(* CODESYS project LuPumping_v3_42.project

Project tree, tasks and I/O mapping:
  LocalDevice : CODESYS Control for Raspberry Pi SL, 3S - Smart Software Solutions GmbH, version 3.5.16.0
    application Application
      libraries: Standard, * (System); VisuDialogs, * (System); SysMem, * (System); SysTimeRtc, * (System); SysRtc23, 3.5.13.0 (System); BASIC, * (OSCAT); CmpBitmapPool, * (System); Util, * (System)
      task VISU_TASK (cyclic, interval 4 ms, priority 31) calls VisuElems.Visu_Prg
      task EtherCAT_Task (cyclic, interval t#4ms, priority 1) calls EtherCAT_Master.EtherCAT_Task
      task MAIN (cyclic, interval t#20ms, priority 1) calls PLC_PRG
      global variables GVL
      Symbols
      Visu_Pages/
        visualisation Visualization_10
        visualisation Visualization_30
        visualisation Visualization_20
        visualisation Visualization_11
        image pool ImagePool
        visualisation Visualization_40
        image pool ImagePool_Presets
        visualisation Visualization_31
      Struct/
        data type ST_ControllerData
        data type ST_ModbusRegister
        data type ST_EtherCATData
        data type ST_PumpingData
        data type ST_PumpingData_HMI
        data type ST_PresetLU
        data type ST_OutBuffer
      program PLC_PRG [ST]
      program _00_Initialization [ST]
      program _01_Comms [ST]
      program _02_Ctrl [ST]
      program _03_daq_setup [ST]
      program _04_daq_input [ST]
      program _05_daq_output [ST]
      program _06_hmi [ST]
    I²C
    GPIOs_A_B : GPIOs A/B, 3S - Smart Software Solutions GmbH, version 3.5.11.0 (disabled)
        unmapped channels: digital inputs (GPIO0..GPIO31), digital outputs (GPIO0..GPIO31)
    SPI
    EtherCAT_Master : EtherCAT Master, 3S - Smart Software Solutions GmbH, version 3.5.16.0
        settings: NetworkName = 'eth0'; NetworkName = "eth0"; SelectNetworkByName = True; SrcAddress1 = 47143; SrcAddress2 = 3947725782
      EK1101 : EK1101 EtherCAT Coupler (2A E-Bus, ID switch), Beckhoff Automation GmbH & Co. KG, order no. EK1101, version Revision=16#00120000
          settings: StationAlias = 0
          unmapped channels: ID
        EL2502_3 : EL2502 2Ch. PWM output, 24V, Beckhoff Automation GmbH & Co. KG, order no. EL2502, version Revision=16#001A0000
            settings: StationAlias = 0
            output Application.GVL.EthCAT.PumpPWM_INT16[5] : UINT  // PWM output
            output Application.GVL.EthCAT.PumpPWM_INT16[6] : UINT  // PWM output
        EL2502_1 : EL2502 2Ch. PWM output, 24V, Beckhoff Automation GmbH & Co. KG, order no. EL2502, version Revision=16#001A0000
            settings: StationAlias = 0; RxTxPdo.NumberofExcludes = 2; RxTxPdo.NumberofEntries = 1; RxTxPdo.Index = 16#1600; RxTxPdo.Fixed = True; RxTxPdo.Mandatory = False; RxTxPdo.Virtual = False; RxTxPdo.Sm = 2; RxTxPdo.Su = 2; RxTxPdo.Name = 'PWM Outputs Channel 1'; RxTxPdo.DependOnSlot = False; RxTxPdo.DependOnSlotGroup = False; RxTxPdo.OverwrittenByModule = False; Exclude = [16#1602,16#1604]; PWM output.Index = 16#7000; PWM output.SubIndex = 17; PWM output.Size = 16; PWM output.Offset = 0; PWM output.DependOnSlot = False; PWM output.DependOnSlotGroup = False; RxTxPdo.NumberofExcludes = 2; RxTxPdo.NumberofEntries = 1; RxTxPdo.Index = 16#1601; RxTxPdo.Fixed = True; RxTxPdo.Mandatory = False; RxTxPdo.Virtual = False; RxTxPdo.Sm = 2; RxTxPdo.Su = 2; RxTxPdo.Name = 'PWM Outputs Channel 2'; RxTxPdo.DependOnSlot = False; RxTxPdo.DependOnSlotGroup = False; RxTxPdo.OverwrittenByModule = False; Exclude = [16#1603,16#1605]; PWM output.Index = 16#7010; PWM output.SubIndex = 17; PWM output.Size = 16; PWM output.Offset = 0; PWM output.DependOnSlot = False; PWM output.DependOnSlotGroup = False; RxTxPdo.NumberofExcludes = 2;
              RxTxPdo.NumberofEntries = 2; RxTxPdo.Index = 16#1602; RxTxPdo.Fixed = True; RxTxPdo.Mandatory = False; RxTxPdo.Virtual = False; RxTxPdo.Sm = -1; RxTxPdo.Su = -1; RxTxPdo.Name = 'PWM Outputs Channel 1'; RxTxPdo.DependOnSlot = False; RxTxPdo.DependOnSlotGroup = False; RxTxPdo.OverwrittenByModule = False; Exclude = [16#1600,16#1604]; PWM output.Index = 16#7000; PWM output.SubIndex = 17; PWM output.Size = 16; PWM output.Offset = 0; PWM output.DependOnSlot = False; PWM output.DependOnSlotGroup = False; PWM period.Index = 16#7000; PWM period.SubIndex = 18; PWM period.Size = 16; PWM period.Offset = 0; PWM period.DependOnSlot = False; PWM period.DependOnSlotGroup = False; RxTxPdo.NumberofExcludes = 2; RxTxPdo.NumberofEntries = 2; RxTxPdo.Index = 16#1603; RxTxPdo.Fixed = True; RxTxPdo.Mandatory = False; RxTxPdo.Virtual = False; RxTxPdo.Sm = -1; RxTxPdo.Su = -1; RxTxPdo.Name = 'PWM Outputs Channel 2'; RxTxPdo.DependOnSlot = False; RxTxPdo.DependOnSlotGroup = False; RxTxPdo.OverwrittenByModule = False; Exclude = [16#1601,16#1605]; PWM output.Index = 16#7010; PWM output.SubIndex = 17; PWM output.Size = 16;
              PWM output.Offset = 0; PWM output.DependOnSlot = False; PWM output.DependOnSlotGroup = False; PWM period.Index = 16#7010; PWM period.SubIndex = 18; PWM period.Size = 16; PWM period.Offset = 0; PWM period.DependOnSlot = False; PWM period.DependOnSlotGroup = False; RxTxPdo.NumberofExcludes = 2; RxTxPdo.NumberofEntries = 2; RxTxPdo.Index = 16#1604; RxTxPdo.Fixed = True; RxTxPdo.Mandatory = False; RxTxPdo.Virtual = False; RxTxPdo.Sm = -1; RxTxPdo.Su = -1; RxTxPdo.Name = 'PWM Outputs Channel 1'; RxTxPdo.DependOnSlot = False; RxTxPdo.DependOnSlotGroup = False; RxTxPdo.OverwrittenByModule = False; Exclude = [16#1600,16#1602]; PWM output.Index = 16#7000; PWM output.SubIndex = 17; PWM output.Size = 16; PWM output.Offset = 0; PWM output.DependOnSlot = False; PWM output.DependOnSlotGroup = False; PWM period 1Hz.Index = 16#7000; PWM period 1Hz.SubIndex = 19; PWM period 1Hz.Size = 32; PWM period 1Hz.Offset = 0; PWM period 1Hz.DependOnSlot = False; PWM period 1Hz.DependOnSlotGroup = False; RxTxPdo.NumberofExcludes = 2; RxTxPdo.NumberofEntries = 2; RxTxPdo.Index = 16#1605; RxTxPdo.Fixed = True; RxTxPdo.Mandatory = False; RxTxPdo.Virtual = False;
              RxTxPdo.Sm = -1; RxTxPdo.Su = -1; RxTxPdo.Name = 'PWM Outputs Channel 2'; RxTxPdo.DependOnSlot = False; RxTxPdo.DependOnSlotGroup = False; RxTxPdo.OverwrittenByModule = False; Exclude = [16#1601,16#1603]; PWM output.Index = 16#7010; PWM output.SubIndex = 17; PWM output.Size = 16; PWM output.Offset = 0; PWM output.DependOnSlot = False; PWM output.DependOnSlotGroup = False; PWM period 1Hz.Index = 16#7010; PWM period 1Hz.SubIndex = 19; PWM period 1Hz.Size = 32; PWM period 1Hz.Offset = 0; PWM period 1Hz.DependOnSlot = False; PWM period 1Hz.DependOnSlotGroup = False; PWM output.Name = 'PWM output'; PWM output.DataType = 'UINT'; PWM output.Default = ''; PWM output.Comment = ''; PWM output.Name = 'PWM output'; PWM output.DataType = 'UINT'; PWM output.Default = ''; PWM output.Comment = ''; PWM output.Name = 'PWM output'; PWM output.DataType = 'UINT'; PWM output.Default = ''; PWM output.Comment = ''; PWM period.Name = 'PWM period'; PWM period.DataType = 'UINT'; PWM period.Default = ''; PWM period.Comment = ''; PWM output.Name = 'PWM output'; PWM output.DataType = 'UINT'; PWM output.Default = ''; PWM output.Comment = ''; PWM period.Name = 'PWM period';
              PWM period.DataType = 'UINT'; PWM period.Default = ''; PWM period.Comment = ''; PWM output.Name = 'PWM output'; PWM output.DataType = 'UINT'; PWM output.Default = ''; PWM output.Comment = ''; PWM period 1Hz.Name = 'PWM period 1Hz'; PWM period 1Hz.DataType = 'UDINT'; PWM period 1Hz.Default = ''; PWM period 1Hz.Comment = ''; PWM output.Name = 'PWM output'; PWM output.DataType = 'UINT'; PWM output.Default = ''; PWM output.Comment = ''; PWM period 1Hz.Name = 'PWM period 1Hz'; PWM period 1Hz.DataType = 'UDINT'; PWM period 1Hz.Default = ''; PWM period 1Hz.Comment = ''
            output Application.GVL.EthCAT.PumpPWM_INT16[1] : UINT  // PWM output
            output Application.GVL.EthCAT.PumpPWM_INT16[2] : UINT  // PWM output
        EL2502_2 : EL2502 2Ch. PWM output, 24V, Beckhoff Automation GmbH & Co. KG, order no. EL2502, version Revision=16#001A0000
            settings: StationAlias = 0
            output Application.GVL.EthCAT.PumpPWM_INT16[3] : UINT  // PWM output
            output Application.GVL.EthCAT.PumpPWM_INT16[4] : UINT  // PWM output
        EL3048 : EL3048 8Ch. Ana. Input 0-20mA, Beckhoff Automation GmbH & Co. KG, order no. EL3048, version Revision=16#00140000
            settings: StationAlias = 0
            input  Application.GVL.EthCAT.Flow2_INT16[1] : INT  // Value
            input  Application.GVL.EthCAT.Flow2_INT16[2] : INT  // Value
            input  Application.GVL.EthCAT.Flow2_INT16[3] : INT  // Value
            input  Application.GVL.EthCAT.Conductivity_INT16 : INT  // Value
            input  Application.GVL.EthCAT.DeltaP2_INT16[1] : INT  // Value
            input  Application.GVL.EthCAT.DeltaP2_INT16[2] : INT  // Value
            unmapped channels: Status__Underrange, Status__Overrange, Status__Limit 1, Status__Limit 1, Status__Limit 2, Status__Limit 2, Status__Error, ---, ---, ---, ---, ---, ---, ---, Status__TxPDO State, Status__TxPDO Toggle, Status__Underrange, Status__Overrange, Status__Limit 1, Status__Limit 1, Status__Limit 2, Status__Limit 2, Status__Error, ---, ---, ---, ---, ---, ---, ---, Status__TxPDO State, Status__TxPDO Toggle, Status__Underrange, Status__Overrange, Status__Limit 1, Status__Limit 1, Status__Limit 2, Status__Limit 2, Status__Error, ---,
              ---, ---, ---, ---, ---, ---, Status__TxPDO State, Status__TxPDO Toggle, Status__Underrange, Status__Overrange, Status__Limit 1, Status__Limit 1, Status__Limit 2, Status__Limit 2, Status__Error, ---, ---, ---, ---, ---, ---, ---, Status__TxPDO State, Status__TxPDO Toggle, Status__Underrange, Status__Overrange, Status__Limit 1, Status__Limit 1, Status__Limit 2, Status__Limit 2, Status__Error, ---, ---, ---, ---, ---, ---, ---, Status__TxPDO State, Status__TxPDO Toggle,
              Status__Underrange, Status__Overrange, Status__Limit 1, Status__Limit 1, Status__Limit 2, Status__Limit 2, Status__Error, ---, ---, ---, ---, ---, ---, ---, Status__TxPDO State, Status__TxPDO Toggle, Status__Underrange, Status__Overrange, Status__Limit 1, Status__Limit 1, Status__Limit 2, Status__Limit 2, Status__Error, ---, ---, ---, ---, ---, ---, ---, Status__TxPDO State, Status__TxPDO Toggle, Value, Status__Underrange, Status__Overrange, Status__Limit 1, Status__Limit 1, Status__Limit 2, Status__Limit 2, Status__Error,
              ---, ---, ---, ---, ---, ---, ---, Status__TxPDO State, Status__TxPDO Toggle, Value
        EL4008 : EL4008 8Ch. Ana. Output 0-10V, 12bit, Beckhoff Automation GmbH & Co. KG, order no. EL4008, version Revision=16#00140000
            settings: StationAlias = 0
            output Application.GVL.EthCAT.ValveOD_INT16[1] : INT  // Analog output
            output Application.GVL.EthCAT.ValveOD_INT16[2] : INT  // Analog output
            output Application.GVL.EthCAT.VPPE_INT16 : INT  // Analog output
            output Application.GVL.EthCAT.ValveOD_INT16[3] : INT  // Analog output
            output Application.GVL.EthCAT.ValveOD_INT16[4] : INT  // Analog output
            unmapped channels: Analog output, Analog output, Analog output
        EL2008 : EL2008 8Ch. Dig. Output 24V, 0.5A, Beckhoff Automation GmbH & Co. KG, order no. EL2008, version Revision=16#00120000
            settings: StationAlias = 0
            output Application.GVL.EthCAT.Valve3_ON[1] : BIT  // Output
            output Application.GVL.EthCAT.Valve3_ON[2] : BIT  // Output
            output Application.GVL.EthCAT.Valve3_ON[3] : BIT  // Output
            output Application.GVL.EthCAT.Valve3_ON[4] : BIT  // Output
            output Application.GVL.EthCAT.Valve3_ON[5] : BIT  // Output
            output Application.GVL.EthCAT.Valve3_ON[6] : BIT  // Output
            output Application.GVL.EthCAT.Valve3_ON[7] : BIT  // Output
            output Application.GVL.EthCAT.Valve3_ON[8] : BIT  // Output
        EL2008_1 : EL2008 8Ch. Dig. Output 24V, 0.5A, Beckhoff Automation GmbH & Co. KG, order no. EL2008, version Revision=16#00120000
            settings: StationAlias = 0
            output Application.GVL.EthCAT.Valve3_ON[9] : BIT  // Output
            output Application.GVL.EthCAT.Valve3_ON[10] : BIT  // Output
            unmapped channels: Output, Output, Output, Output, Output, Output
        EL3068_1 : EL3068 8Ch. Ana. Input 0-10V, Beckhoff Automation GmbH & Co. KG, order no. EL3068, version Revision=16#00140000
            settings: StationAlias = 0
            input  Application.GVL.EthCAT.Temperature1_INT16[1] : INT  // Value
            input  Application.GVL.EthCAT.Pressure1_INT16[1] : INT  // Value
            input  Application.GVL.EthCAT.Temperature1_INT16[2] : INT  // Value
            input  Application.GVL.EthCAT.Pressure1_INT16[2] : INT  // Value
            input  Application.GVL.EthCAT.Temperature1_INT16[3] : INT  // Value
            input  Application.GVL.EthCAT.Pressure1_INT16[3] : INT  // Value
            input  Application.GVL.EthCAT.Temperature1_INT16[4] : INT  // Value
            input  Application.GVL.EthCAT.Pressure1_INT16[4] : INT  // Value
            unmapped channels: Status__Underrange, Status__Overrange, Status__Limit 1, Status__Limit 1, Status__Limit 2, Status__Limit 2, Status__Error, ---, ---, ---, ---, ---, ---, ---, Status__TxPDO State, Status__TxPDO Toggle, Status__Underrange, Status__Overrange, Status__Limit 1, Status__Limit 1, Status__Limit 2, Status__Limit 2, Status__Error, ---, ---, ---, ---, ---, ---, ---, Status__TxPDO State, Status__TxPDO Toggle, Status__Underrange, Status__Overrange, Status__Limit 1, Status__Limit 1, Status__Limit 2, Status__Limit 2, Status__Error, ---,
              ---, ---, ---, ---, ---, ---, Status__TxPDO State, Status__TxPDO Toggle, Status__Underrange, Status__Overrange, Status__Limit 1, Status__Limit 1, Status__Limit 2, Status__Limit 2, Status__Error, ---, ---, ---, ---, ---, ---, ---, Status__TxPDO State, Status__TxPDO Toggle, Status__Underrange, Status__Overrange, Status__Limit 1, Status__Limit 1, Status__Limit 2, Status__Limit 2, Status__Error, ---, ---, ---, ---, ---, ---, ---, Status__TxPDO State, Status__TxPDO Toggle,
              Status__Underrange, Status__Overrange, Status__Limit 1, Status__Limit 1, Status__Limit 2, Status__Limit 2, Status__Error, ---, ---, ---, ---, ---, ---, ---, Status__TxPDO State, Status__TxPDO Toggle, Status__Underrange, Status__Overrange, Status__Limit 1, Status__Limit 1, Status__Limit 2, Status__Limit 2, Status__Error, ---, ---, ---, ---, ---, ---, ---, Status__TxPDO State, Status__TxPDO Toggle, Status__Underrange, Status__Overrange, Status__Limit 1, Status__Limit 1, Status__Limit 2, Status__Limit 2, Status__Error, ---,
              ---, ---, ---, ---, ---, ---, Status__TxPDO State, Status__TxPDO Toggle
        EL3068 : EL3068 8Ch. Ana. Input 0-10V, Beckhoff Automation GmbH & Co. KG, order no. EL3068, version Revision=16#00140000
            settings: StationAlias = 0
            input  Application.GVL.EthCAT.Level_INT16[1] : INT  // Value
            input  Application.GVL.EthCAT.Level_INT16[2] : INT  // Value
            input  Application.GVL.EthCAT.Level_INT16[3] : INT  // Value
            input  Application.GVL.EthCAT.Level_INT16[4] : INT  // Value
            unmapped channels: Status__Underrange, Status__Overrange, Status__Limit 1, Status__Limit 1, Status__Limit 2, Status__Limit 2, Status__Error, ---, ---, ---, ---, ---, ---, ---, Status__TxPDO State, Status__TxPDO Toggle, Status__Underrange, Status__Overrange, Status__Limit 1, Status__Limit 1, Status__Limit 2, Status__Limit 2, Status__Error, ---, ---, ---, ---, ---, ---, ---, Status__TxPDO State, Status__TxPDO Toggle, Status__Underrange, Status__Overrange, Status__Limit 1, Status__Limit 1, Status__Limit 2, Status__Limit 2, Status__Error, ---,
              ---, ---, ---, ---, ---, ---, Status__TxPDO State, Status__TxPDO Toggle, Status__Underrange, Status__Overrange, Status__Limit 1, Status__Limit 1, Status__Limit 2, Status__Limit 2, Status__Error, ---, ---, ---, ---, ---, ---, ---, Status__TxPDO State, Status__TxPDO Toggle, Status__Underrange, Status__Overrange, Status__Limit 1, Status__Limit 1, Status__Limit 2, Status__Limit 2, Status__Error, ---, ---, ---, ---, ---, ---, ---, Status__TxPDO State, Status__TxPDO Toggle,
              Value, Status__Underrange, Status__Overrange, Status__Limit 1, Status__Limit 1, Status__Limit 2, Status__Limit 2, Status__Error, ---, ---, ---, ---, ---, ---, ---, Status__TxPDO State, Status__TxPDO Toggle, Value, Status__Underrange, Status__Overrange, Status__Limit 1, Status__Limit 1, Status__Limit 2, Status__Limit 2, Status__Error, ---, ---, ---, ---, ---, ---, ---, Status__TxPDO State, Status__TxPDO Toggle, Value, Status__Underrange, Status__Overrange, Status__Limit 1, Status__Limit 1, Status__Limit 2,
              Status__Limit 2, Status__Error, ---, ---, ---, ---, ---, ---, ---, Status__TxPDO State, Status__TxPDO Toggle, Value
    Onewire
    SoftMotion General Axis Pool
    Camera device
      <Empty>
    Ethernet : Ethernet, 3S - Smart Software Solutions GmbH, version 3.5.16.0
        settings: IPAddress = [192,168,100,42]; SubnetMask = [255,255,255,0]; GatewayAddress = [192,168,0,1]; MACAddress = [16#00,16#00,16#00,16#00,16#00,16#00]; NetworkInterfaceName = 'eth1'; NetworkInterfaceName = "eth1"; SaveCommunicationSettings = FALSE
      ModbusTCP_Server_CCU : ModbusTCP Slave Device, 3S - Smart Software Solutions GmbH, version 3.5.16.0
          input  Application.GVL.ModbusCCU.REGIN : ARRAY[0..19] OF WORD  // Inputs
          output Application.GVL.ModbusCCU.REGOUT : ARRAY[0..19] OF WORD  // Outputs
      ModbusTCP_Server_LU : ModbusTCP Slave Device, 3S - Smart Software Solutions GmbH, version 3.5.16.0
          settings: Port = 503
          input  Application.GVL.ModbusLU.REGIN : ARRAY[0..19] OF WORD  // Inputs
          output Application.GVL.ModbusLU.REGOUT : ARRAY[0..19] OF WORD  // Outputs
  text list GlobalTextList
  GlobalImagePool
  5ce3da45-db07-42e7-a21c-a00fff4ed8f6|\\ES.AAU.DK\Users\jvl\Pictures\HMI\valve_off.png
  5ce3da45-db07-42e7-a21c-a00fff4ed8f6|ImagePool\valve_off.png
  5ce3da45-db07-42e7-a21c-a00fff4ed8f6|ImagePool\Background.png
  5ce3da45-db07-42e7-a21c-a00fff4ed8f6|ImagePool\Preset15.png
*)

// LocalDevice/Application/Struct/ST_ControllerData
TYPE ST_ControllerData :
STRUCT
//LU STATUS
	
    nStatus_CtrlMode			: INT := 1;	// Control Mode Selection
	nStatus_CtrlModeAUX			: INT := 1;
	nStatus_LockSetup_ON		: BOOL;	// LU configuration is blocked.
	
	nStatus_LevelControl_ON		: BOOL;
	nStatus_TankLevel_Max		: BOOL;
	nStatus_TankLevel_Min		: BOOL;
	
    nStatus_Warning          	: BIT;
	nStatus_CommAlarm		 	: BIT;
	nStatus_user				: STRING := 'ad';
	nStatus_pass				: STRING := '0';
	
//PRESETS
	Idx_Preset				: INT :=0;
	Idx_PresetHMI			: INT :=0;

(*Preset configuration of the LU
	-ID 		(INT) - Identification Number for each preset.
	-Name 	(STR) - 
	-Valve_Preset (WORD) - 10 bits of the WORD are used as a mask to turn on/off the valves for the different configurations:
		Bit9(V_51), Bit8(V_42),
 		Bit7(V_41)	Bit6(V_32)	Bit5(V_22)	Bit4(V_21)
		Bit3(V_14)	Bit2(V_13)	Bit1(V_12)	Bit0(V_11)
				
	-Component_Enable(BYTE) - 4 bits of the BYTE 
		Bit7(V_22)	Bit6(V_21)	Bit5(V_12)	Bit4(Pu_Gr3)
		Bit3(Pu_Gr2)	Bit2(Pu_Gr1)	Bit1(V_51 Bit0(V_31)
*)

PresetLU	 : ARRAY[0..16] OF ST_PresetLU:=[(ID:=0 	,Name:='All_Closed'			,Valve_Preset:=2#00_0000_0000 , Component_Enabled := 2#0000_0000),
											(ID:=1 		,Name:='All_Open'			,Valve_Preset:=2#11_1111_1111 , Component_Enabled := 2#0001_1111),
											(ID:=2 		,Name:='WSS + Aux_Supply'	,Valve_Preset:=2#10_0100_0100 , Component_Enabled := 2#0000_1101),
											(ID:=3 		,Name:='WSS2 + Aux_Supply'	,Valve_Preset:=2#10_0111_0011 , Component_Enabled := 2#0000_1101),
											(ID:=4 		,Name:='Tank1 + Aux_Supply'	,Valve_Preset:=2#10_0011_0001 , Component_Enabled := 2#0000_1001),
											(ID:=5 		,Name:='Tank2'				,Valve_Preset:=2#01_0011_0000 , Component_Enabled := 2#0001_0001),
											(ID:=6 		,Name:='Mix 1'				,Valve_Preset:=2#00_1100_0100 , Component_Enabled := 2#0000_0110),
											(ID:=7 		,Name:='Mix 2'				,Valve_Preset:=2#10_1100_0100 , Component_Enabled := 2#0000_1100),
											(ID:=8 		,Name:='Mix 3'				,Valve_Preset:=2#01_0100_0100 , Component_Enabled := 2#0001_0110),
											(ID:=9 		,Name:='Mix 4'				,Valve_Preset:=2#01_0000_0100 , Component_Enabled := 2#0001_0011),
											(ID:=10		,Name:='Mix5a'				,Valve_Preset:=2#10_1111_0010 , Component_Enabled := 2#0000_1100),
											(ID:=11		,Name:='Mix5b'				,Valve_Preset:=2#10_1011_1010 , Component_Enabled := 2#0000_1100),
											(ID:=12 	,Name:='WWS1 + Aux_Supply'	,Valve_Preset:=2#10_0110_0001 , Component_Enabled := 2#0100_1100),
											(ID:=13 	,Name:='WWS2 + Aux_Supply'	,Valve_Preset:=2#10_0111_0001 , Component_Enabled := 2#0000_1101),
											(ID:=14		,Name:='WWS3 + Aux_Supply'	,Valve_Preset:=2#10_0100_0000 , Component_Enabled := 2#1110_1100),
											(ID:=15		,Name:='WWS4 + 2 Supply'	,Valve_Preset:=2#10_1111_0001 , Component_Enabled := 2#1110_1111) ];										
//MODBUS REGISTERS	
	Modbus	: ST_ModbusRegister;
	
//LU DATA
	Data	: ST_PumpingData;
	HMI_Data : ST_PumpingData_HMI;

END_STRUCT
END_TYPE

// LocalDevice/Application/Struct/ST_ModbusRegister
TYPE ST_ModbusRegister :
STRUCT
	REGIN	: ARRAY[0..19] OF WORD;
	REGOUT	: ARRAY[0..19] OF WORD;	
	COIL_IN : ARRAY[0..20] OF BOOL;
END_STRUCT
END_TYPE

// LocalDevice/Application/Struct/ST_EtherCATData
TYPE ST_EtherCATData :
STRUCT
(*Mapping of the EtherCAT modules with system variables scale_INT16(bits)*)

//I/O Ethercat slave modules
(*Input Variables*)
	Flow2_INT16				: ARRAY[1..3] OF WORD;
	Temperature1_INT16		: ARRAY[1..4]OF WORD;
	Pressure1_INT16			: ARRAY[1..4]OF WORD;
	DeltaP2_INT16			: ARRAY[1..2] OF WORD;
	Conductivity_INT16		: WORD;
	Level_INT16				: ARRAY[1..4] OF WORD;
(*Output Variables*)
	PumpPWM_INT16			: ARRAY[1..6] OF WORD;
	ValveOD_INT16 			: ARRAY[1..4] OF WORD;
	Valve3_ON				: ARRAY[1..10] OF BOOL;
	VPPE_INT16				: WORD; // Air pressure reference for air control VPPE [0-10V]
	
END_STRUCT
END_TYPE

// LocalDevice/Application/Struct/ST_PumpingData
TYPE ST_PumpingData :
STRUCT
	
	(*============= LU ============== UINT = REAL x 1000*)	
	
(*Input Variables*)	
	
	Q2_11, Q2_12, Q2_51 : UINT;
	C1 : UINT;
	dP2_in, dP2_ex, TankLevel_in, TankLevel_ex 	: UINT; // Tank level in % 
	dP2_in_MAX, dP2_ex_MAX, dP2_in_MIN, dP2_ex_MIN : UINT;
	T31, T32, T33, T51 : UINT;
	P31, P32, P33, P51 : UINT;
	L_11, L_12, L_21, L_22 : UINT;
	Sewer_DN : UINT;
	Q_estim_L22 : UINT;
	
(*Output Variables *)		
	V3_11_ON, V3_12_ON, V3_13_ON, V3_14_ON, V3_21_ON, V3_22_ON, V3_32_ON, V3_41_ON, V3_42_ON, V3_52_ON : BOOL;
	ValveOD_31, ValveOD_51, ValveOD_61,ValveOD_71 				: UINT;
	Pu_1, Pu_2, Pu_3, Pu_4, Pu_5, Pu_6	: UINT;	
	Pu_1_fb, Pu_2_fb, Pu_3_fb, Pu_4_fb, Pu_5_fb, Pu_6_fb	: UINT;	
	VPPE 	: UINT;
	
(*Offset of the variables - after scale*)
	Offset_F2				: ARRAY[1..5] OF WORD;
	Offset_C				: WORD;
	Offset_T1				: ARRAY[1..12] OF WORD;
	Offset_P1				: ARRAY[1..12] OF WORD;
	Offset_dP2				: ARRAY[1..2] OF WORD;	
	Offset_L				: ARRAY[1..4] OF UINT;
	
END_STRUCT
END_TYPE

// LocalDevice/Application/Struct/ST_PumpingData_HMI
TYPE ST_PumpingData_HMI :
STRUCT
	
	(*============= HMI ==============*)
	
(*Input Variables*)	
	
	Q2_11, Q2_12, Q2_51 : REAL;
	C1 : REAL;
	dP2_in, dP2_ex, TankFill_in, TankFill_ex 	: REAL;
	T31, T32, T33, T51 : REAL;
	P31, P32, P33, P51 : REAL;
	L_11, L_12, L_21, L_22 : REAL;
	Q_estim_L22 : REAL;
	
(*Output Variables *)		
	ValveOD_31, ValveOD_51, ValveOD_61,ValveOD_71 				: REAL;
	ValveOD_31_input, ValveOD_51_input, ValveOD_61_input,ValveOD_71_input	: REAL;
	Pu_1, Pu_2, Pu_3, Pu_4, Pu_5, Pu_6	: REAL;
	Pu_1_input, Pu_2_input, Pu_3_input, Pu_4_input, Pu_5_input, Pu_6_input	: REAL;
	
	Pu_1_fb, Pu_2_fb, Pu_3_fb, Pu_4_fb, Pu_5_fb, Pu_6_fb	: REAL;	
	VPPE 	: REAL;
	
	ManMode, LUmode, CCUmode : BOOL;
	
	F_TankLevel_in_MAX, F_TankLevel_in_MIN, F_TankLevel_ex_MAX, F_TankLevel_ex_MIN : BOOL;
	
	
	
	
END_STRUCT
END_TYPE

// LocalDevice/Application/Struct/ST_PresetLU
TYPE ST_PresetLU :
STRUCT
	
	ID				: UINT		:=99;
	Name			: STRING 	:='PresetName';
	AuxSupply_Mode	: BOOL 		:= FALSE;
	Valve_Preset	: WORD 		:= 2#0000_0000_0000_0000;
	Component_Enabled	: BYTE	:= 2#0000_0000; // 2#0000_Va51.Gr2.Va31.Gr1
	
END_STRUCT
END_TYPE

// LocalDevice/Application/Struct/ST_OutBuffer
TYPE ST_OutBuffer :
STRUCT
	ValveOD_31 : WORD; 
	ValveOD_51 : WORD;
	ValveOD_61 : WORD;
	ValveOD_71 : WORD;
		
	Pu_1 : WORD;
	Pu_2 : WORD;
	Pu_3 : WORD;
	Pu_4 : WORD;
	Pu_5 : WORD;
	Pu_6 : WORD;
	
	Valve_12_ON : BOOL;
	Valve_13_ON : BOOL;
	Valve_21_ON : BOOL;
	Valve_22_ON : BOOL;	
	
END_STRUCT
END_TYPE

// LocalDevice/Application/GVL
{attribute 'qualified_only'}
VAR_GLOBAL
	
(*Controller Variables*)
	myLU		: ST_ControllerData;
	EthCAT 		: ST_EtherCATData;
	ModbusCCU	: ST_ModbusRegister;		// Remote modbust to Central Control Unit
	ModbusLU 	: ST_ModbusRegister; 		// Localhost modbus to LU client

(*Variables - DAQ*);	
	i, j		: INT; 

	MaxRange_INT16 		: UINT := 32767; //number of bits in a positive value
	MaxRange_UINT16 	: UINT := 65535;
	MinRange_INT16		: UINT := 6554; // Min nr. of bits for [2-10]V [4-20]mA - 32767*(2/10)
	
(*Variables - HMI*)	
	Plot_ON		: ARRAY[1..50] OF BOOL;
	DynamicImgID	: STRING;
	
(*COMMUNICATION SETUP*)
    TON1: STD.TON; // Communication Timeout
	TON1_timeset: TIME := T#5S;
	ModbusCnt: WORD;
	ModbusCnt_Old: WORD;

(* AUXILIARY VARIABLES FOR CONTROL *)
	F_TankInfeed_ON : BOOL;
	F_TankOutfeed_ex_ON : BOOL;
	
	F_TankOutfeed_in_ON : BOOL;
END_VAR

// LocalDevice/Application/PLC_PRG
PROGRAM PLC_PRG
VAR
	F_init : BOOL := FALSE;
END_VAR

(*Main Routine*)

IF F_init = FALSE THEN
	_00_Initialization();
	F_init := TRUE;
END_IF

_01_Comms();

_02_Ctrl();

_03_daq_setup();

_04_daq_input();

_05_daq_output();

_06_hmi();

END_PROGRAM

// LocalDevice/Application/_00_Initialization
PROGRAM _00_Initialization
VAR
	EK1101_ID: UINT := 0;
END_VAR

(*Initialization of the LU*)

(*Initialize the status of the controller.*)
	GVL.MyLU.nStatus_CommAlarm := FALSE;
	GVL.MyLU.nStatus_LockSetup_ON := TRUE;
	GVL.MyLU.nStatus_Warning := 0;
	GVL.myLU.nStatus_LevelControl_ON := TRUE;

(*Initialize offset variables *)

//Pressure 1
	GVL.MyLU.Data.Offset_P1[1] := 0;
	GVL.MyLU.Data.Offset_P1[2] := 0;
	GVL.MyLU.Data.Offset_P1[3] := 0;
	GVL.MyLU.Data.Offset_P1[4] := 0;

//Diff. pressure.
	GVL.MyLU.Data.Offset_dP2[1] := 0;//100
	GVL.MyLU.Data.Offset_dP2[2] := 0 ;	//507
	
// Tank Level
	GVL.myLU.Data.dP2_ex_MAX := 564;
	GVL.myLU.Data.dP2_in_MAX := 768;
	GVL.myLU.Data.dP2_in_MIN := 100;
	GVL.myLU.Data.dP2_in_MIN := 100;
	
//Flow 2
	GVL.MyLU.Data.Offset_F2[1] := 0;
	GVL.MyLU.Data.Offset_F2[2] := 0;
	GVL.MyLU.Data.Offset_F2[3] := 0;
	GVL.MyLU.Data.Offset_F2[4] := 0;
	GVL.MyLU.Data.Offset_F2[5] := 0;
//Conductivity
	GVL.MyLU.Data.Offset_C := 0;

// Level

	GVL.myLU.Data.Offset_L[1] := 0;
	GVL.myLU.Data.Offset_L[2] := 0;
	GVL.myLU.Data.Offset_L[3] := 0;
	GVL.myLU.Data.Offset_L[4] := 0;
	
// Diameter
	GVL.myLU.Data.Sewer_DN := 50;
	
// 

(*Init Preset configuration*)

END_PROGRAM

// LocalDevice/Application/_01_Comms
PROGRAM _01_Comms
VAR
END_VAR

(* Communication 
	Mapping of the Registers with MyLU.Data
*)

CASE GVL.myLU.nStatus_CtrlMode OF
	1:
	GVL.MyLU.Modbus.REGIN 	:= GVL.ModbusCCU.REGIN;		//INPUT - Read input values from MODBUS input registers
		GVL.ModbusCCU.REGOUT	:= GVL.MyLU.Modbus.REGOUT;		//OUTPUT - Write output values to MODBUS holding registers		
	2: // Auto - Local - Use port nr 503 for local Modbus comms 
		GVL.MyLU.Modbus.REGIN := GVL.ModbusLU.REGIN;
		GVL.ModbusLU.REGOUT:= GVL.MyLU.Modbus.REGOUT;	
	3:  // Auto - Remote - Use port nr 502 for remote Modbus comms
		GVL.MyLU.Modbus.REGIN 	:= GVL.ModbusCCU.REGIN;		//INPUT - Read input values from MODBUS input registers
		GVL.ModbusCCU.REGOUT	:= GVL.MyLU.Modbus.REGOUT;		//OUTPUT - Write output values to MODBUS holding registers		
END_CASE

//MODBUS TIMEOUT

IF GVL.MyLU.nStatus_CtrlMode = (1 OR 2 OR 3) THEN
	// Mapping of the DAQ to output data array
		
	// Mapping of Inputs
	
	// Timeout
	GVL.ModbusCnt := GVL.MyLU.Modbus.REGIN[0];
	GVL.TON1(IN:= GVL.ModbusCnt = GVL.ModbusCnt_Old,PT:= GVL.TON1_timeset);
	GVL.ModbusCnt_Old := GVL.ModbusCnt;
	
	IF GVL.TON1.Q = TRUE THEN
		GVL.MyLU.nStatus_CommAlarm := TRUE;
	END_IF

END_IF

END_PROGRAM

// LocalDevice/Application/_02_Ctrl
PROGRAM _02_Ctrl

(*Control LU*)

(*Tank Level Control*)

IF GVL.mylu.nStatus_LevelControl_ON THEN
	
(*High Level Limit with hysteresis*)
	IF (GVL.myLU.Data.dP2_ex > 560) OR (GVL.myLU.Data.dP2_in > 850) THEN
		GVL.F_TankInfeed_ON := FALSE;
	ELSIF (GVL.myLU.Data.dP2_ex < 450) OR (GVL.myLU.Data.dP2_in < 750) THEN
		GVL.F_TankInfeed_ON := TRUE;
	END_IF 

(*Low Level Limit with hysteresis*)
(*External Tank Outfeed*)
	IF (GVL.myLU.Data.dP2_ex < 90)  THEN
		GVL.F_TankOutfeed_ex_ON := FALSE;
	ELSIF (GVL.myLU.Data.dP2_ex > 100) THEN
		GVL.F_TankOutfeed_ex_ON := TRUE;
	END_IF
(*Internal Tank Outfeed*)
	IF  (GVL.myLU.Data.dP2_in < 150) THEN
		GVL.F_TankOutfeed_in_ON := FALSE;
	ELSIF (GVL.myLU.Data.dP2_in > 250) THEN
		GVL.F_TankOutfeed_in_ON := TRUE;
	END_IF 
	
ELSE
	GVL.F_TankInfeed_ON  := TRUE;
	GVL.F_TankOutfeed_ex_ON := TRUE;
	GVL.F_TankOutfeed_in_ON := TRUE;
END_IF

END_PROGRAM

// LocalDevice/Application/_03_daq_setup
PROGRAM _03_daq_setup
VAR
	OutBuffer			: ST_OutBuffer;	
	
END_VAR

(*  ============= CONTROL MODE SELECTION: ===================== 
	1 = Manual
	2 = Local
	3 = Remote *)
	
(* Predefined configurations*)
GVL.i := GVL.MyLU.Idx_PresetHMI;
GVL.j := GVL.MyLU.Idx_Preset;

(*Mode Selection*)


CASE GVL.MyLU.nStatus_CtrlMode OF
	1: //Manual )
		OutBuffer.ValveOD_31 := REAL_TO_UINT(GVL.MyLU.HMI_Data.ValveOD_31_input*100);
		OutBuffer.ValveOD_51 := REAL_TO_UINT(GVL.MyLU.HMI_Data.ValveOD_51_input*100);	
		OutBuffer.ValveOD_61 := REAL_TO_UINT(GVL.MyLU.HMI_Data.ValveOD_61_input*100);
		OutBuffer.ValveOD_71 := REAL_TO_UINT(GVL.MyLU.HMI_Data.ValveOD_71_input*100);
		
		OutBuffer.Pu_1 := REAL_TO_UINT(GVL.MyLU.HMI_Data.Pu_1_input*100);
		OutBuffer.Pu_2 := REAL_TO_UINT(GVL.MyLU.HMI_Data.Pu_2_input*100);
		OutBuffer.Pu_3 := REAL_TO_UINT(GVL.MyLU.HMI_Data.Pu_3_input*100);
		OutBuffer.Pu_4 := REAL_TO_UINT(GVL.MyLU.HMI_Data.Pu_4_input*100);
		OutBuffer.Pu_5 := REAL_TO_UINT(GVL.MyLU.HMI_Data.Pu_5_input*100);
		OutBuffer.Pu_6 := REAL_TO_UINT(GVL.MyLU.HMI_Data.Pu_6_input*100);
		
		GVL.myLU.Modbus.REGOUT[0] := GVL.MyLU.Data.L_11 ;
		GVL.myLU.Modbus.REGOUT[1] := GVL.MyLU.Data.L_12 ;
		GVL.myLU.Modbus.REGOUT[2] := GVL.MyLU.Data.L_21 ;
		GVL.myLU.Modbus.REGOUT[3] := GVL.MyLU.Data.L_22 ;
		
	2..3: // Auto - Local - Use port nr 503 for local Modbus comms 
	
		OutBuffer.ValveOD_31 := GVL.MyLU.Modbus.REGIN[1];
		OutBuffer.ValveOD_51 := GVL.MyLU.Modbus.REGIN[2];	
		OutBuffer.ValveOD_61 := GVL.MyLU.Modbus.REGIN[3];
		OutBuffer.ValveOD_71 := GVL.MyLU.Modbus.REGIN[4];
	
		OutBuffer.Pu_1 := GVL.MyLU.Modbus.REGIN[5];
		OutBuffer.Pu_2 := GVL.MyLU.Modbus.REGIN[6];
		OutBuffer.Pu_3 := GVL.MyLU.Modbus.REGIN[7];
		OutBuffer.Pu_4 := GVL.MyLU.Modbus.REGIN[8];
		OutBuffer.Pu_5 := GVL.MyLU.Modbus.REGIN[9];
		OutBuffer.Pu_6 := GVL.MyLU.Modbus.REGIN[10];	
		
		GVL.MyLU.Data.Q_estim_L22 := GVL.myLU.Modbus.REGIN[11];

		
		GVL.myLU.Modbus.REGOUT[0] := GVL.MyLU.Data.P31;
		GVL.myLU.Modbus.REGOUT[1] := GVL.MyLU.Data.P32;
		GVL.myLU.Modbus.REGOUT[2] := GVL.MyLU.Data.P33;
		GVL.myLU.Modbus.REGOUT[3] := GVL.MyLU.Data.P51;
		GVL.myLU.Modbus.REGOUT[4] := GVL.MyLU.Data.dP2_ex;
		GVL.myLU.Modbus.REGOUT[5] := GVL.MyLU.Data.dP2_in;
		
		GVL.myLU.Modbus.REGOUT[6] := GVL.MyLU.Data.T31 ; 
		GVL.myLU.Modbus.REGOUT[7] := GVL.MyLU.Data.T32 ;  //
		GVL.myLU.Modbus.REGOUT[8] := GVL.MyLU.Data.T33 ; 
		GVL.myLU.Modbus.REGOUT[9] := GVL.MyLU.Data.T51 ;
		
		GVL.myLU.Modbus.REGOUT[10] := GVL.MyLU.Data.Q2_11 ;
		GVL.myLU.Modbus.REGOUT[11] := GVL.MyLU.Data.Q2_12 ;
		GVL.myLU.Modbus.REGOUT[12] := GVL.MyLU.Data.Q2_51 ;
		GVL.myLU.Modbus.REGOUT[13] := GVL.MyLU.Data.C1;
 
		GVL.myLU.Modbus.REGOUT[14] := GVL.MyLU.Data.L_11 ;
		GVL.myLU.Modbus.REGOUT[15] := GVL.MyLU.Data.L_12 ;
		GVL.myLU.Modbus.REGOUT[16] := GVL.MyLU.Data.L_21 ;
		GVL.myLU.Modbus.REGOUT[17] := GVL.MyLU.Data.L_22 ;

ELSE 
	GVL.MyLU.nStatus_CtrlMode := 1;
END_CASE
	
		
(* ============= PRESET SETUP =============== 

Failsafe operation - Enable LU components

*)

//ENABLE CONTROLLABLE VALVES

IF GVL.MyLU.PresetLU[GVL.j].Component_Enabled.0 THEN
	GVL.MyLU.Data.ValveOD_31 := OutBuffer.ValveOD_31;
ELSE
	GVL.MyLU.Data.ValveOD_31 := 0;
END_IF
IF GVL.MyLU.PresetLU[GVL.j].Component_Enabled.1  THEN
	GVL.MyLU.Data.ValveOD_51 := OutBuffer.ValveOD_51;
ELSE
	GVL.MyLU.Data.ValveOD_51 := 0;
END_IF

IF GVL.F_TankInfeed_ON THEN
	GVL.MyLU.Data.ValveOD_61 := OutBuffer.ValveOD_61;
	GVL.MyLU.Data.ValveOD_71 := OutBuffer.ValveOD_71;
ELSE
	GVL.MyLU.Data.ValveOD_61 := 0;
	GVL.MyLU.Data.ValveOD_71 := 0;
END_IF	
	
//ENABLE PUMPS (Pu1, Pu2, Pu3)  - (Pu4, Pu5) - (Pu&)

IF GVL.MyLU.PresetLU[GVL.j].Component_Enabled.2 THEN
	GVL.MyLU.Data.Pu_1 := OutBuffer.Pu_1;
	GVL.MyLU.Data.Pu_2 := OutBuffer.Pu_2;
	GVL.MyLU.Data.Pu_3 := OutBuffer.Pu_3;
ELSE
	GVL.MyLU.Data.Pu_1 := 0;
	GVL.MyLU.Data.Pu_2 := 0;
	GVL.MyLU.Data.Pu_3 := 0;	
END_IF

IF GVL.MyLU.PresetLU[GVL.j].Component_Enabled.3 THEN
	GVL.MyLU.Data.Pu_4 := OutBuffer.Pu_4;
	GVL.MyLU.Data.Pu_5 := OutBuffer.Pu_5;
ELSE
	GVL.MyLU.Data.Pu_4 := 0;
	GVL.MyLU.Data.Pu_5 := 0;
END_IF

IF GVL.MyLU.PresetLU[GVL.j].Component_Enabled.4 THEN
	GVL.MyLU.Data.Pu_6 := OutBuffer.Pu_6;
ELSE
	GVL.MyLU.Data.Pu_6 := 0;
END_IF

//ENABLE SHUT OFF VALVES:

//V_11
IF GVL.F_TankInfeed_ON THEN
	GVL.myLU.Data.V3_11_ON := GVL.MyLU.PresetLU[GVL.j].Valve_Preset.0;
ELSE
	GVL.myLU.Data.V3_11_ON := FALSE;
END_IF

//V_12
IF GVL.F_TankInfeed_ON AND GVL.MyLU.PresetLU[GVL.j].Component_Enabled.5 THEN
	GVL.myLU.Data.V3_12_ON := OutBuffer.Valve_12_ON;
ELSIF GVL.F_TankInfeed_ON AND NOT GVL.MyLU.PresetLU[GVL.j].Component_Enabled.5 THEN
	GVL.myLU.Data.V3_12_ON := GVL.MyLU.PresetLU[GVL.j].Valve_Preset.1;
ELSE
	GVL.myLU.Data.V3_12_ON := FALSE;	
END_IF

//V_13
IF GVL.MyLU.PresetLU[GVL.j].Component_Enabled.5 THEN
	GVL.myLU.Data.V3_13_ON := OutBuffer.Valve_13_ON;
ELSE
	GVL.myLU.Data.V3_13_ON := GVL.MyLU.PresetLU[GVL.j].Valve_Preset.2;
END_IF

//V_14
GVL.myLU.Data.V3_14_ON := GVL.MyLU.PresetLU[GVL.j].Valve_Preset.3;

//V_21	
IF GVL.F_TankOutfeed_ex_ON AND GVL.MyLU.PresetLU[GVL.j].Component_Enabled.6 THEN
	GVL.myLU.Data.V3_21_ON := OutBuffer.Valve_21_ON;
ELSIF GVL.F_TankOutfeed_ex_ON AND NOT GVL.MyLU.PresetLU[GVL.j].Component_Enabled.6 THEN
	GVL.myLU.Data.V3_21_ON := GVL.MyLU.PresetLU[GVL.j].Valve_Preset.4;
ELSE
	GVL.myLU.Data.V3_21_ON := FALSE;	
END_IF

//V_22
IF GVL.F_TankOutfeed_in_ON AND GVL.MyLU.PresetLU[GVL.j].Component_Enabled.7 THEN
	GVL.myLU.Data.V3_22_ON := OutBuffer.Valve_22_ON;
ELSIF GVL.F_TankOutfeed_in_ON AND NOT GVL.MyLU.PresetLU[GVL.j].Component_Enabled.7 THEN
	GVL.myLU.Data.V3_22_ON := GVL.MyLU.PresetLU[GVL.j].Valve_Preset.5;
ELSE
	GVL.myLU.Data.V3_22_ON := 0;	
END_IF


//V_32
GVL.myLU.Data.V3_32_ON := GVL.MyLU.PresetLU[GVL.j].Valve_Preset.6;

//V_41
GVL.myLU.Data.V3_41_ON := GVL.MyLU.PresetLU[GVL.j].Valve_Preset.7;

//V_42
GVL.myLU.Data.V3_42_ON := GVL.MyLU.PresetLU[GVL.j].Valve_Preset.8;

//V_52
GVL.myLU.Data.V3_52_ON := GVL.MyLU.PresetLU[GVL.j].Valve_Preset.9;

END_PROGRAM

// LocalDevice/Application/_04_daq_input
PROGRAM _04_daq_input
VAR
	(*Variables - DAQ*);
	LIN_TRAFO	: ARRAY[1..18] OF UTIL.LIN_TRAFO;

END_VAR

(*DATA ACQUISITION MAPPING AND LINEALIZATION 
Data conversion of the raw I/O values to...
	FROM	INT16 (Raw value from Beckhoff module)	- 12 bit (16 bit presentation, incl. sign )
	TO	 	REAL(UINT) (Scaled value *100)      *)
	
(*========== INPUTs ========*)

(*Pressure 1 - Grundfos [...to  meterH2O(x100)]*)
//P31 	- 	
	LIN_TRAFO[1](IN:=GVL.EthCAT.Pressure1_INT16[1], IN_MIN:=0, IN_MAX:=GVL.MaxRange_INT16, OUT_MIN :=0, OUT_MAX:=1.6*9.82*100);
	GVL.MyLU.Data.P31 := REAL_TO_WORD(LIN_TRAFO[1].OUT) - GVL.MyLU.Data.Offset_P1[1];
//P32
	LIN_TRAFO[2](IN:=GVL.EthCAT.Pressure1_INT16[2], IN_MIN:=0, IN_MAX:=GVL.MaxRange_INT16, OUT_MIN:=0, OUT_MAX:=1.6*9.82*100);
	GVL.MyLU.Data.P32 := REAL_TO_WORD(LIN_TRAFO[2].OUT) - GVL.MyLU.Data.Offset_P1[2];
//P33
	LIN_TRAFO[3](IN:=GVL.EthCAT.Pressure1_INT16[3], IN_MIN:=0, IN_MAX:=GVL.MaxRange_INT16, OUT_MIN:=0, OUT_MAX:=1.6*9.82*100);
	GVL.MyLU.Data.P33 := REAL_TO_WORD(LIN_TRAFO[3].OUT) - GVL.MyLU.Data.Offset_P1[3];
//P51	-	Pressure 1 - Grundfos  [...to  meterH2O(x100)]
	LIN_TRAFO[4](IN:=GVL.EthCAT.Pressure1_INT16[4],	IN_MIN:=0, IN_MAX:=GVL.MaxRange_INT16,	OUT_MIN:=0, OUT_MAX:=1.6*9.82*100);
	GVL.MyLU.Data.P51 := REAL_TO_WORD(LIN_TRAFO[4].OUT) - GVL.MyLU.Data.Offset_P1[4];
	
(*Differential Pressure [ ...to meters. e.g 2.5meterH2O(x100)]*)

//dP2 ext	
	LIN_TRAFO[5](IN:= GVL.EthCAT.DeltaP2_INT16[1],IN_MIN:= GVL.MinRange_INT16 ,IN_MAX:= GVL.MaxRange_INT16,OUT_MIN:= 0, OUT_MAX:=2000);
	GVL.MyLU.Data.dP2_ex:= REAL_TO_WORD(LIN_TRAFO[5].OUT);
//dP2 int	
	LIN_TRAFO[6](IN:= GVL.EthCAT.DeltaP2_INT16[2],IN_MIN:= GVL.MinRange_INT16 ,IN_MAX:= GVL.MaxRange_INT16,OUT_MIN:= 0, OUT_MAX:=2000);
	GVL.MyLU.Data.dP2_in := REAL_TO_WORD(LIN_TRAFO[6].OUT);
	
(*Temperature [... to Celsious degrees(x100) ]*)		
// T31 
	LIN_TRAFO[7](IN:= GVL.EthCAT.Temperature1_INT16[1], IN_MIN:=0, IN_MAX:= GVL.MaxRange_INT16, OUT_MIN:=0, OUT_MAX:=100*100);
	GVL.MyLU.Data.T31 := REAL_TO_WORD(LIN_TRAFO[7].OUT) -  GVL.MyLU.Data.Offset_T1[1];
//T32 
	LIN_TRAFO[8](IN:= GVL.EthCAT.Temperature1_INT16[2], IN_MIN:=0, IN_MAX:= GVL.MaxRange_INT16, OUT_MIN:=0, OUT_MAX:=100*100);
	GVL.MyLU.Data.T32 := REAL_TO_WORD(LIN_TRAFO[8].OUT) -  GVL.MyLU.Data.Offset_T1[2];
//T33
	LIN_TRAFO[9](IN:= GVL.EthCAT.Temperature1_INT16[3], IN_MIN:=0, IN_MAX:= GVL.MaxRange_INT16, OUT_MIN:=0, OUT_MAX:=100*100);
	GVL.MyLU.Data.T33 := REAL_TO_WORD(LIN_TRAFO[9].OUT) -  GVL.MyLU.Data.Offset_T1[3];
//T51
	LIN_TRAFO[10](IN:= GVL.EthCAT.Temperature1_INT16[4], IN_MIN:=0, IN_MAX:= GVL.MaxRange_INT16, OUT_MIN:=0, OUT_MAX:=100*100);
	GVL.MyLU.Data.T51 := REAL_TO_WORD(LIN_TRAFO[10].OUT) -  GVL.MyLU.Data.Offset_T1[4];
	
(*FLow3 [ ..to l/min(x100)]*)	
//Q1_11 
	LIN_TRAFO[11](IN:= GVL.EthCAT.Flow2_INT16[1],IN_MIN:= GVL.MinRange_INT16, IN_MAX:= GVL.MaxRange_INT16, OUT_MIN:=0, OUT_MAX:=100*100);
	GVL.MyLU.Data.Q2_11 := REAL_TO_WORD(LIN_TRAFO[11].OUT) - GVL.MyLU.Data.Offset_F2[1];
//Q1_12
	LIN_TRAFO[12](IN:= GVL.EthCAT.Flow2_INT16[2],IN_MIN:= GVL.MinRange_INT16, IN_MAX:= GVL.MaxRange_INT16, OUT_MIN:=0, OUT_MAX:=100*100);
	GVL.MyLU.Data.Q2_12 := REAL_TO_WORD(LIN_TRAFO[12].OUT) - GVL.MyLU.Data.Offset_F2[2];
//Q1_51
	LIN_TRAFO[13](IN:= GVL.EthCAT.Flow2_INT16[3],IN_MIN:= GVL.MinRange_INT16, IN_MAX:= GVL.MaxRange_INT16, OUT_MIN:=0, OUT_MAX:=100*100);
	GVL.MyLU.Data.Q2_51 := REAL_TO_WORD(LIN_TRAFO[13].OUT) - GVL.MyLU.Data.Offset_F2[3];


(*Conductivity [... to uS(x100)]*)
// C
	LIN_TRAFO[14](IN:= GVL.EthCAT.Conductivity_INT16,IN_MIN:= GVL.MinRange_INT16, IN_MAX:= GVL.MaxRange_INT16, OUT_MIN:=0, OUT_MAX:=1*100);
	GVL.MyLU.Data.C1 := REAL_TO_WORD(LIN_TRAFO[14].OUT) - GVL.MyLU.Data.Offset_C;

(*Water Level [ ...to mm(x100)]*)

//L_11
	LIN_TRAFO[15](IN:= GVL.EthCAT.Level_INT16[1],IN_MIN:= 100, IN_MAX:= 10800, OUT_MIN:=0, OUT_MAX:=50);
	GVL.MyLU.Data.L_11 := (GVL.MyLU.Data.Sewer_DN - REAL_TO_WORD(LIN_TRAFO[15].OUT)+ GVL.MyLU.Data.Offset_L[1]);
// L_12
	LIN_TRAFO[16](IN:= GVL.EthCAT.Level_INT16[2],IN_MIN:= 100, IN_MAX:= 10800, OUT_MIN:=0, OUT_MAX:=50);
	GVL.MyLU.Data.L_12 := (GVL.MyLU.Data.Sewer_DN - REAL_TO_WORD(LIN_TRAFO[16].OUT)+ GVL.MyLU.Data.Offset_L[2]);
// L_21
	LIN_TRAFO[17](IN:= GVL.EthCAT.Level_INT16[3],IN_MIN:= 100, IN_MAX:= 10800, OUT_MIN:=0, OUT_MAX:=50);
	GVL.MyLU.Data.L_21 := (GVL.MyLU.Data.Sewer_DN - REAL_TO_WORD(LIN_TRAFO[17].OUT)+ GVL.MyLU.Data.Offset_L[3]);
// L_22	
	LIN_TRAFO[18](IN:= GVL.EthCAT.Level_INT16[4],IN_MIN:= 100, IN_MAX:= 10800, OUT_MIN:=0, OUT_MAX:=50);
	GVL.MyLU.Data.L_22 := (GVL.MyLU.Data.Sewer_DN - REAL_TO_WORD(LIN_TRAFO[18].OUT)+ GVL.MyLU.Data.Offset_L[4]);

END_PROGRAM

// LocalDevice/Application/_05_daq_output
PROGRAM _05_daq_output
VAR
	(*Variables - DAQ*);
	LIN_TRAFO	: ARRAY[1..14] OF UTIL.LIN_TRAFO;
END_VAR

(*========== OUTPUTSs ========*)

(*Valve OD - Belimo valve %(x100)  *)

//V1_11	-  
	LIN_TRAFO[1](IN:= GVL.MyLU.Data.ValveOD_31,IN_MIN:= 0,IN_MAX:=100*100,OUT_MIN := GVL.MinRange_INT16, OUT_MAX:=GVL.MaxRange_INT16);
	GVL.EthCAT.ValveOD_INT16[1] := REAL_TO_WORD(LIN_TRAFO[1].OUT);
//V1_12
	LIN_TRAFO[2](IN:= GVL.MyLU.Data.ValveOD_51,IN_MIN:= 0,IN_MAX:=100*100,OUT_MIN := GVL.MinRange_INT16, OUT_MAX:=GVL.MaxRange_INT16);
	GVL.EthCAT.ValveOD_INT16[2] := REAL_TO_WORD(LIN_TRAFO[2].OUT);
//V1_13
	LIN_TRAFO[3](IN:= GVL.MyLU.Data.ValveOD_61,IN_MIN:= 0,IN_MAX:=100*100,OUT_MIN := GVL.MinRange_INT16, OUT_MAX:= GVL.MaxRange_INT16);
	GVL.EthCAT.ValveOD_INT16[3] := REAL_TO_WORD(LIN_TRAFO[3].OUT);
//V1_21
	LIN_TRAFO[4](IN:= GVL.MyLU.Data.ValveOD_71,IN_MIN:= 0,IN_MAX:=100*100,OUT_MIN := GVL.MinRange_INT16, OUT_MAX:= GVL.MaxRange_INT16);
	GVL.EthCAT.ValveOD_INT16[4] := REAL_TO_WORD(LIN_TRAFO[4].OUT);


(*Pump Speed PWM_DC - UPM3 %(x100)
	CONTROL NOTE: <= 10% Max Speed
			>10 / 84<= Variable speed
			>84 / 91 <= Minimum speed
			>91/95 Hysteresys area On/Off
			>95 / 100 Standby mode: Off *)	

// Pump1  
	LIN_TRAFO[5](IN:= GVL.MyLU.Data.Pu_1,IN_MIN:= 0,IN_MAX:=100*100,OUT_MIN := GVL.MaxRange_INT16, OUT_MAX:= 0);
	GVL.EthCAT.PumpPWM_INT16[1] := REAL_TO_WORD(LIN_TRAFO[5].OUT);
// Pump 2 
	LIN_TRAFO[6](IN:= GVL.MyLU.Data.Pu_2,IN_MIN:= 0,IN_MAX:=100*100,OUT_MIN := GVL.MaxRange_INT16, OUT_MAX:= 0);
	GVL.EthCAT.PumpPWM_INT16[2] := REAL_TO_WORD(LIN_TRAFO[6].OUT);
// Pump 3 
	LIN_TRAFO[7](IN:= GVL.MyLU.Data.Pu_3,IN_MIN:= 0,IN_MAX:=100*100,OUT_MIN := GVL.MaxRange_INT16, OUT_MAX:= 0);
	GVL.EthCAT.PumpPWM_INT16[3] := REAL_TO_WORD(LIN_TRAFO[7].OUT);
// Pump 4 
	LIN_TRAFO[8](IN:= GVL.MyLU.Data.Pu_4,IN_MIN:= 0,IN_MAX:=100*100,OUT_MIN := GVL.MaxRange_INT16, OUT_MAX:= 0);
	GVL.EthCAT.PumpPWM_INT16[4] := REAL_TO_WORD(LIN_TRAFO[8].OUT);
// Pump 5 
	LIN_TRAFO[9](IN:= GVL.MyLU.Data.Pu_5,IN_MIN:= 0,IN_MAX:=100*100,OUT_MIN := GVL.MaxRange_INT16, OUT_MAX:= 0);
	GVL.EthCAT.PumpPWM_INT16[5] := REAL_TO_WORD(LIN_TRAFO[9].OUT);
// Pump 6 
	LIN_TRAFO[10](IN:= GVL.MyLU.Data.Pu_6,IN_MIN:= 0,IN_MAX:=100*100,OUT_MIN := GVL.MaxRange_INT16, OUT_MAX:= 0);
	GVL.EthCAT.PumpPWM_INT16[6] := REAL_TO_WORD(LIN_TRAFO[10].OUT);

	
(*Air pressure ref for tank - FESTO VPPE [From meters x100..] *)
// VPPE reference. for tank air pressure.
	LIN_TRAFO[11](IN:= GVL.MyLU.Data.VPPE,IN_MIN:= 0,IN_MAX:=2*10*100,OUT_MIN := 0, OUT_MAX:=GVL.MaxRange_INT16);
	GVL.EthCAT.VPPE_INT16:= REAL_TO_WORD(LIN_TRAFO[11].OUT);
		
(*Preset configurations of the LU *)

//Shut Off Valves

	GVL.EthCAT.Valve3_ON[1] := GVL.myLU.Data.V3_11_ON;
	GVL.EthCAT.Valve3_ON[2] := GVL.myLU.Data.V3_12_ON;
	GVL.EthCAT.Valve3_ON[3] := GVL.myLU.Data.V3_13_ON;
	GVL.EthCAT.Valve3_ON[4] := GVL.myLU.Data.V3_14_ON;
	GVL.EthCAT.Valve3_ON[5] := GVL.myLU.Data.V3_21_ON;
	GVL.EthCAT.Valve3_ON[6] := GVL.myLU.Data.V3_22_ON;
	GVL.EthCAT.Valve3_ON[7] := GVL.myLU.Data.V3_32_ON;
	GVL.EthCAT.Valve3_ON[8] := GVL.myLU.Data.V3_41_ON;
	GVL.EthCAT.Valve3_ON[9] := GVL.myLU.Data.V3_42_ON;
	GVL.EthCAT.Valve3_ON[10] := GVL.myLU.Data.V3_52_ON;

END_PROGRAM

// LocalDevice/Application/_06_hmi
PROGRAM _06_hmi
VAR
END_VAR

(*HMI CONTROL*)

// Pressure [ ... to meters.]
	GVL.MyLU.HMI_Data.P31 := UINT_TO_REAL(GVL.MyLU.Data.P31)/100;
	GVL.MyLU.HMI_Data.P32 := UINT_TO_REAL(GVL.MyLU.Data.P32)/100;
	GVL.MyLU.HMI_Data.P33 := UINT_TO_REAL(GVL.MyLU.Data.P33)/100;	
	GVL.MyLU.HMI_Data.P51 := UINT_TO_REAL(GVL.MyLU.Data.P51)/100;
		
// Temperature [... to Celsious degrees.]	
	GVL.MyLU.HMI_Data.T31 := UINT_TO_REAL(GVL.MyLU.Data.T31)/100;
	GVL.MyLU.HMI_Data.T32 := UINT_TO_REAL(GVL.MyLU.Data.T32)/100;
	GVL.MyLU.HMI_Data.T33 := UINT_TO_REAL(GVL.MyLU.Data.T33)/100;
	GVL.MyLU.HMI_Data.T51 := UINT_TO_REAL(GVL.MyLU.Data.T51)/100;

// FLow1 [ ..to l/min]
	GVL.MyLU.HMI_Data.Q2_11 := UINT_TO_REAL(GVL.MyLU.Data.Q2_11)/100;
	GVL.MyLU.HMI_Data.Q2_12 := UINT_TO_REAL(GVL.MyLU.Data.Q2_12)/100;
	GVL.MyLU.HMI_Data.Q2_51 := UINT_TO_REAL(GVL.MyLU.Data.Q2_51)/100;
	
// Conductivity [... to uS]
	GVL.MyLU.HMI_Data.C1 := UINT_TO_REAL(GVL.MyLU.Data.C1)/100;

// Differential pressure
	GVL.MyLU.HMI_Data.dP2_in := UINT_TO_REAL(GVL.MyLU.Data.dP2_in);
	GVL.MyLU.HMI_Data.dP2_ex := UINT_TO_REAL(GVL.MyLU.Data.dP2_ex);	
	
// Valves 
	GVL.MyLU.HMI_Data.ValveOD_31 := UINT_TO_REAL(GVL.MyLU.Data.ValveOD_31)/100;
	GVL.MyLU.HMI_Data.ValveOD_51 := UINT_TO_REAL(GVL.MyLU.Data.ValveOD_51)/100;
	GVL.MyLU.HMI_Data.ValveOD_61 := UINT_TO_REAL(GVL.MyLU.Data.ValveOD_61)/100;
	GVL.MyLU.HMI_Data.ValveOD_71 := UINT_TO_REAL(GVL.MyLU.Data.ValveOD_71)/100;
	
// Pumps	
	GVL.MyLU.HMI_Data.Pu_1 := UINT_TO_REAL(GVL.MyLU.Data.Pu_1)/100;
	GVL.MyLU.HMI_Data.Pu_2 := UINT_TO_REAL(GVL.MyLU.Data.Pu_2)/100;
	GVL.MyLU.HMI_Data.Pu_3 := UINT_TO_REAL(GVL.MyLU.Data.Pu_3)/100;
	GVL.MyLU.HMI_Data.Pu_4 := UINT_TO_REAL(GVL.MyLU.Data.Pu_4)/100;
	GVL.MyLU.HMI_Data.Pu_5 := UINT_TO_REAL(GVL.MyLU.Data.Pu_5)/100;
	GVL.MyLU.HMI_Data.Pu_6 := UINT_TO_REAL(GVL.MyLU.Data.Pu_6)/100;
	
// Level	
	GVL.MyLU.HMI_Data.L_11 := UINT_TO_REAL(GVL.MyLU.Data.L_11);
	GVL.MyLU.HMI_Data.L_12 := UINT_TO_REAL(GVL.MyLU.Data.L_12);
	GVL.MyLU.HMI_Data.L_21 := UINT_TO_REAL(GVL.MyLU.Data.L_21);
	GVL.MyLU.HMI_Data.L_22 := UINT_TO_REAL(GVL.MyLU.Data.L_22);
	
	GVL.MyLU.HMI_Data.Q_estim_L22 := UINT_TO_REAL(GVL.MyLU.Data.Q_estim_L22)/100;
	
// Air pressure
	GVL.MyLU.HMI_Data.VPPE := UINT_TO_REAL(GVL.MyLU.Data.VPPE)/100;
	
	
// Lamp indicator at configuration page.	
CASE GVL.MyLU.nStatus_CtrlMode OF
	1:
		GVL.MyLU.HMI_Data.ManMode := TRUE;
		GVL.MyLU.HMI_Data.LUmode := FALSE;
		GVL.MyLU.HMI_Data.CCUmode := FALSE;
	2:
		GVL.MyLU.HMI_Data.ManMode := FALSE;
		GVL.MyLU.HMI_Data.LUmode := TRUE;
		GVL.MyLU.HMI_Data.CCUmode := FALSE;
	3:
		GVL.MyLU.HMI_Data.ManMode := FALSE;
		GVL.MyLU.HMI_Data.LUmode := FALSE;
		GVL.MyLU.HMI_Data.CCUmode := TRUE;
END_CASE

// Lamps for tank level indication

IF GVL.F_TankInfeed_ON = FALSE THEN
	GVL.myLU.HMI_Data.F_TankLevel_ex_MAX := TRUE;
ELSIF GVL.F_TankOutfeed_ex_ON = FALSE THEN
	GVL.myLU.HMI_Data.F_TankLevel_ex_MIN := TRUE;
	GVL.myLU.HMI_Data.F_TankLevel_in_MIN := TRUE;
ELSE
	GVL.myLU.HMI_Data.F_TankLevel_ex_MAX := FALSE;
	GVL.myLU.HMI_Data.F_TankLevel_ex_MIN := FALSE;
	GVL.myLU.HMI_Data.F_TankLevel_in_MIN := FALSE;
END_IF

	IF (GVL.myLU.Data.dP2_in > 655) THEN
		GVL.myLU.HMI_Data.F_TankLevel_in_MAX := TRUE;
	ELSIF (GVL.myLU.Data.dP2_ex < 655)  THEN
		GVL.myLU.HMI_Data.F_TankLevel_in_MAX := FALSE;
	END_IF 

	

(*Dynamic Image ID for LU Presets*)

	GVL.DynamicImgID := STD.CONCAT('ImagePool_Presets.',INT_TO_STRING(GVL.MyLU.Idx_PresetHMI));

END_PROGRAM

// LocalDevice/Application/Visu_Pages/Visualization_10
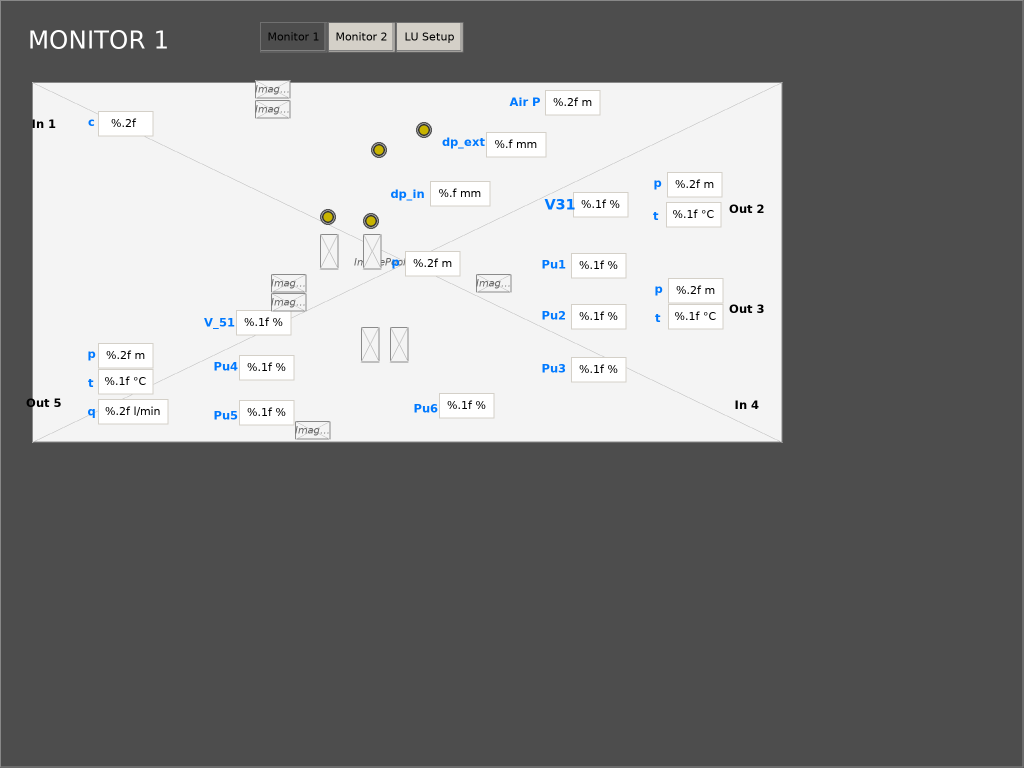
VISUALIZATION Visualization_10  // 1024x768, background image ImagePool.Background
    Image (32,82 750x360), image: ImagePool.Main_bold
    Label (25,25 180x30), "MONITOR 1"
    Button (260,22 67x30), "Monitor 1"
        OnMouseUp:  Assign=Visualization_10, Type=Assignment
    Button (328,22 67x30), "Monitor 2"
        OnMouseUp:  Assign=Visualization_11, Type=Assignment
    Button (396,22 67x30), "LU Setup"
        OnMouseUp:  Assign=Visualization_20, Type=Assignment
    Label (24,113 40x22), "In 1"
    Label (24,392 40x22), "Out 5"
    Textfield (98,399 70x25), "%.2f l/min", text variable: GVL.myLU.HMI_Data.Q2_51
    Label (80,399 23x25), "q"
    Textfield (668,278 55x25), "%.2f m", text variable: GVL.myLU.HMI_Data.P33
    Textfield (668,304 55x25), "%.1f °C", text variable: GVL.myLU.HMI_Data.T32
    Label (646,274 25x30), "p"
    Label (645,303 26x30), "t"
    Label (507,87 36x30), "Air P"
    Textfield (239,400 55x25), "%.1f %", text variable: GVL.myLU.HMI_Data.Pu_5
    Label (207,403 38x25), "Pu5"
    Label (727,395 40x20), "In 4"
    Label (727,199 40x20), "Out 2"
    Label (727,299 40x20), "Out 3"
    Label (645,168 25x30), "p"
    Textfield (667,172 55x25), "%.2f m", text variable: GVL.myLU.HMI_Data.P32
    Textfield (666,202 55x25), "%.1f °C", text variable: GVL.myLU.HMI_Data.T31
    Label (643,201 26x30), "t"
    Textfield (573,192 55x25), "%.1f %", text variable: GVL.myLU.HMI_Data.ValveOD_31
    Label (541,192 38x25), "V31"
    Label (207,354 38x25), "Pu4"
    Textfield (239,355 55x25), "%.1f %", text variable: GVL.myLU.HMI_Data.Pu_4
    Label (198,310 43x25), "V_51"
    Textfield (236,310 55x25), "%.1f %", text variable: GVL.myLU.HMI_Data.ValveOD_51
    Textfield (98,111 55x25), "%.2f", text variable: GVL.myLU.HMI_Data.C1
    Label (79,107 25x30), "c"
    Textfield (98,343 55x25), "%.2f m", text variable: GVL.myLU.HMI_Data.P51
    Textfield (98,369 55x25), "%.1f °C", text variable: GVL.myLU.HMI_Data.T51
    Label (79,339 25x30), "p"
    Label (78,368 26x30), "t"
    Label (535,252 38x25), "Pu1"
    Textfield (571,253 55x25), "%.1f %", text variable: GVL.myLU.HMI_Data.Pu_1
    Label (535,303 38x25), "Pu2"
    Textfield (571,304 55x25), "%.1f %", text variable: GVL.myLU.HMI_Data.Pu_2
    Label (535,356 38x25), "Pu3"
    Textfield (571,357 55x25), "%.1f %", text variable: GVL.myLU.HMI_Data.Pu_3
    Textfield (486,132 60x25), "%.f mm", text variable: GVL.myLU.HMI_Data.dP2_ex
    Label (443,127 41x30), "dp_ext"
    Textfield (430,181 60x25), "%.f mm", text variable: GVL.myLU.HMI_Data.dP2_in
    Label (387,179 41x30), "dp_in"
    Textfield (545,90 55x25), "%.2f m", text variable: GVL.myLU.HMI_Data.VPPE
    ImageSwitcher (320,234 18x35), variable: GVL.myLU.Data.V3_21_ON, input disabled if: GVL.MyLU.nStatus_LockSetup_ON, background image: ImagePool.valve_on, image: ImagePool.valve_off, behaviour: TOGGLE
    ImageSwitcher (361,327 18x35), variable: GVL.myLU.Data.V3_41_ON, input disabled if: GVL.MyLU.nStatus_LockSetup_ON, background image: ImagePool.valve_on, image: ImagePool.valve_off, behaviour: TOGGLE
    ImageSwitcher (390,327 18x35), variable: GVL.myLU.Data.V3_42_ON, input disabled if: GVL.MyLU.nStatus_LockSetup_ON, background image: ImagePool.valve_on, image: ImagePool.valve_off, behaviour: TOGGLE
    ImageSwitcher (255,80 35x18), variable: GVL.myLU.Data.V3_11_ON, input disabled if: GVL.MyLU.nStatus_LockSetup_ON, background image: valve_on_h, image: valve_off_h, behaviour: TOGGLE
    ImageSwitcher (255,100 35x18), variable: GVL.myLU.Data.V3_12_ON, input disabled if: GVL.MyLU.nStatus_LockSetup_ON, background image: valve_on_h, image: valve_off_h, behaviour: TOGGLE
    ImageSwitcher (271,274 35x18), variable: GVL.myLU.Data.V3_13_ON, input disabled if: GVL.MyLU.nStatus_LockSetup_ON, background image: valve_on_h, image: valve_off_h, behaviour: TOGGLE
    ImageSwitcher (271,293 35x18), variable: GVL.myLU.Data.V3_14_ON, input disabled if: GVL.MyLU.nStatus_LockSetup_ON, background image: valve_on_h, image: valve_off_h, behaviour: TOGGLE
    ImageSwitcher (476,274 35x18), variable: GVL.myLU.Data.V3_32_ON, input disabled if: GVL.MyLU.nStatus_LockSetup_ON, background image: valve_on_h, image: valve_off_h, behaviour: TOGGLE
    ImageSwitcher (295,421 35x18), variable: GVL.myLU.Data.V3_52_ON, input disabled if: GVL.MyLU.nStatus_LockSetup_ON, background image: valve_on_h, image: valve_off_h, behaviour: TOGGLE
    Lamp1 (370,141 18x18), variable: GVL.myLU.HMI_Data.F_TankLevel_in_MAX, style: Lamp-Lamp1-Yellow
    Lamp1 (415,121 18x18), variable: GVL.myLU.HMI_Data.F_TankLevel_ex_MAX, style: Lamp-Lamp1-Yellow
    Lamp1 (362,212 18x18), variable: GVL.myLU.HMI_Data.F_TankLevel_in_MIN, style: Lamp-Lamp1-Yellow
    Textfield (439,393 55x25), "%.1f %", text variable: GVL.myLU.HMI_Data.Pu_6
    Label (407,396 38x25), "Pu6"
    Lamp1 (319,208 18x18), variable: GVL.myLU.HMI_Data.F_TankLevel_ex_MIN, style: Lamp-Lamp1-Yellow
    ImageSwitcher (363,234 18x35), variable: GVL.myLU.Data.V3_22_ON, input disabled if: GVL.MyLU.nStatus_LockSetup_ON, background image: ImagePool.valve_on, image: ImagePool.valve_off, behaviour: TOGGLE
    Label (383,247 25x30), "p"
    Textfield (405,251 55x25), "%.2f m", text variable: GVL.myLU.HMI_Data.P31
END_VISUALIZATION

// LocalDevice/Application/Visu_Pages/Visualization_30
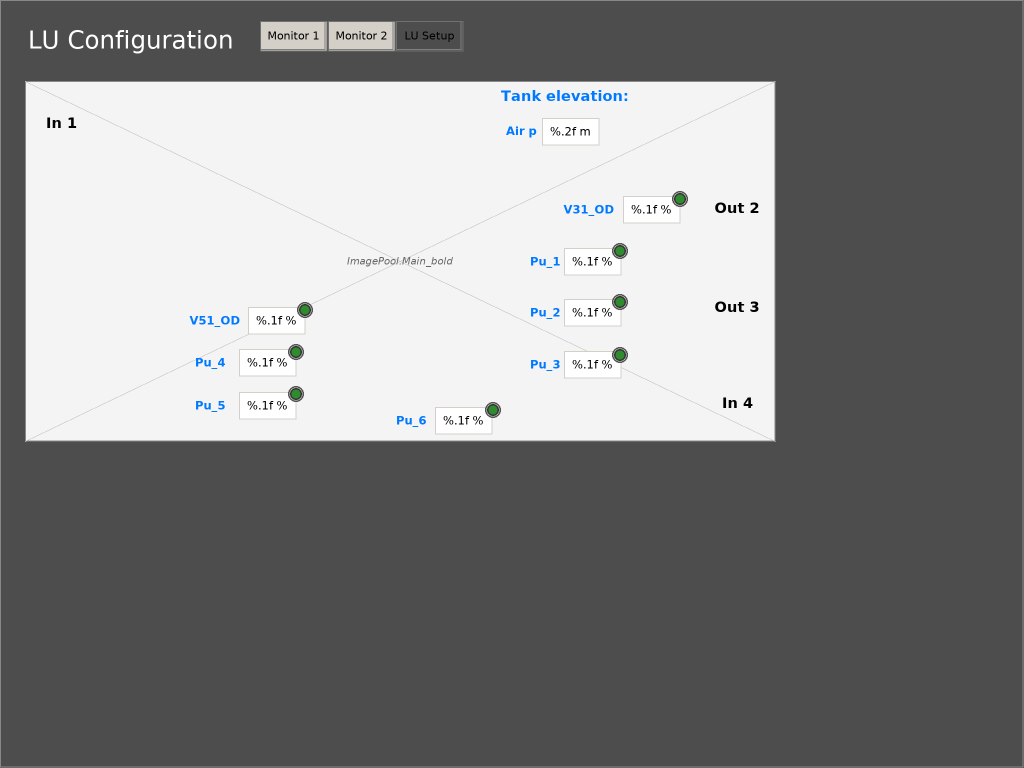
VISUALIZATION Visualization_30  // 1024x768, background image ImagePool.Background
    Label (25,25 318x30), "LU Configuration"
    Button (260,21 67x30), "Monitor 1"
        OnMouseUp:  Assign=Visualization_10, Type=Assignment
    Button (328,21 67x30), "Monitor 2"
        OnMouseUp:  Assign=Visualization_11, Type=Assignment
    Button (396,21 67x30), "LU Setup"
        OnMouseUp:  Assign=Visualization_20, Type=Assignment
    Label (32,391 66x22), "Out 5"
    Image (25,81 750x360), image: ImagePool.Main_bold
    Label (509,81 112x30), "Tank elevation:"
    Textfield (542,118 57x27), "%.2f m", text variable: GVL.myLU.HMI_Data.VPPE
        OnMouseUp: write the text variable via VisuDialogs.Numpad, min 0, max 5, format 0
    Label (494,116 55x30), "Air p"
    Textfield (248,307 57x27), "%.1f %", text variable: GVL.myLU.HMI_Data.ValveOD_51
        OnMouseUp: write GVL.myLU.HMI_Data.ValveOD_51_input via VisuDialogs.Numpad, min 0, max 100, format 0
    Label (185,307 60x27), "V51_OD"
    Textfield (239,349 57x27), "%.1f %", text variable: GVL.myLU.HMI_Data.Pu_4
        OnMouseUp: write GVL.myLU.HMI_Data.Pu_4_input via VisuDialogs.Numpad, min 0, max 100, format 0
    Label (183,349 55x27), "Pu_4"
    Textfield (239,392 57x27), "%.1f %", text variable: GVL.myLU.HMI_Data.Pu_5
        OnMouseUp: write GVL.myLU.HMI_Data.Pu_5_input via VisuDialogs.Numpad, min 0, max 100, format 0
    Label (183,392 55x27), "Pu_5"
    Textfield (564,248 57x27), "%.1f %", text variable: GVL.myLU.HMI_Data.Pu_1
        OnMouseUp: write GVL.myLU.HMI_Data.Pu_1_input via VisuDialogs.Numpad, min 0, max 100, format 0
    Label (518,248 55x27), "Pu_1"
    Textfield (564,299 57x27), "%.1f %", text variable: GVL.myLU.HMI_Data.Pu_2
        OnMouseUp: write GVL.myLU.HMI_Data.Pu_2_input via VisuDialogs.Numpad, min 0, max 100, format 0
    Label (518,299 55x27), "Pu_2"
    Textfield (564,351 57x27), "%.1f %", text variable: GVL.myLU.HMI_Data.Pu_3
        OnMouseUp: write GVL.myLU.HMI_Data.Pu_3_input via VisuDialogs.Numpad, min 0, max 100, format 0
    Label (518,351 55x27), "Pu_3"
    Label (32,112 59x22), "In 1"
    Label (708,392 59x22), "In 4"
    Label (704,197 66x22), "Out 2"
    Label (704,296 66x22), "Out 3"
    Textfield (435,407 57x27), "%.1f %", text variable: GVL.myLU.HMI_Data.Pu_6
        OnMouseUp: write GVL.myLU.HMI_Data.Pu_6_input via VisuDialogs.Numpad, min 0, max 100, format 0
    Label (384,407 55x27), "Pu_6"
    Label (559,196 60x27), "V31_OD"
    Textfield (623,196 57x27), "%.1f %", text variable: GVL.myLU.HMI_Data.ValveOD_31
        OnMouseUp: write GVL.myLU.HMI_Data.ValveOD_31_input via VisuDialogs.Numpad, min 0, max 100, format 0
    Lamp1 (671,190 18x18), variable: GVL.MyLU.PresetLU[GVL.j].Component_Enabled.0, style: Lamp-Lamp1-Green
    Lamp1 (296,301 18x18), variable: GVL.MyLU.PresetLU[GVL.j].Component_Enabled.1, style: Lamp-Lamp1-Green
    Lamp1 (484,401 18x18), variable: GVL.MyLU.PresetLU[GVL.j].Component_Enabled.4, style: Lamp-Lamp1-Green
    Lamp1 (287,343 18x18), variable: GVL.MyLU.PresetLU[GVL.j].Component_Enabled.3, style: Lamp-Lamp1-Green
    Lamp1 (611,242 18x18), variable: GVL.MyLU.PresetLU[GVL.j].Component_Enabled.2, style: Lamp-Lamp1-Green
    Lamp1 (611,293 18x18), variable: GVL.MyLU.PresetLU[GVL.j].Component_Enabled.2, style: Lamp-Lamp1-Green
    Lamp1 (611,346 18x18), variable: GVL.MyLU.PresetLU[GVL.j].Component_Enabled.2, style: Lamp-Lamp1-Green
    Lamp1 (287,385 18x18), variable: GVL.MyLU.PresetLU[GVL.j].Component_Enabled.3, style: Lamp-Lamp1-Green
END_VISUALIZATION

// LocalDevice/Application/Visu_Pages/Visualization_20
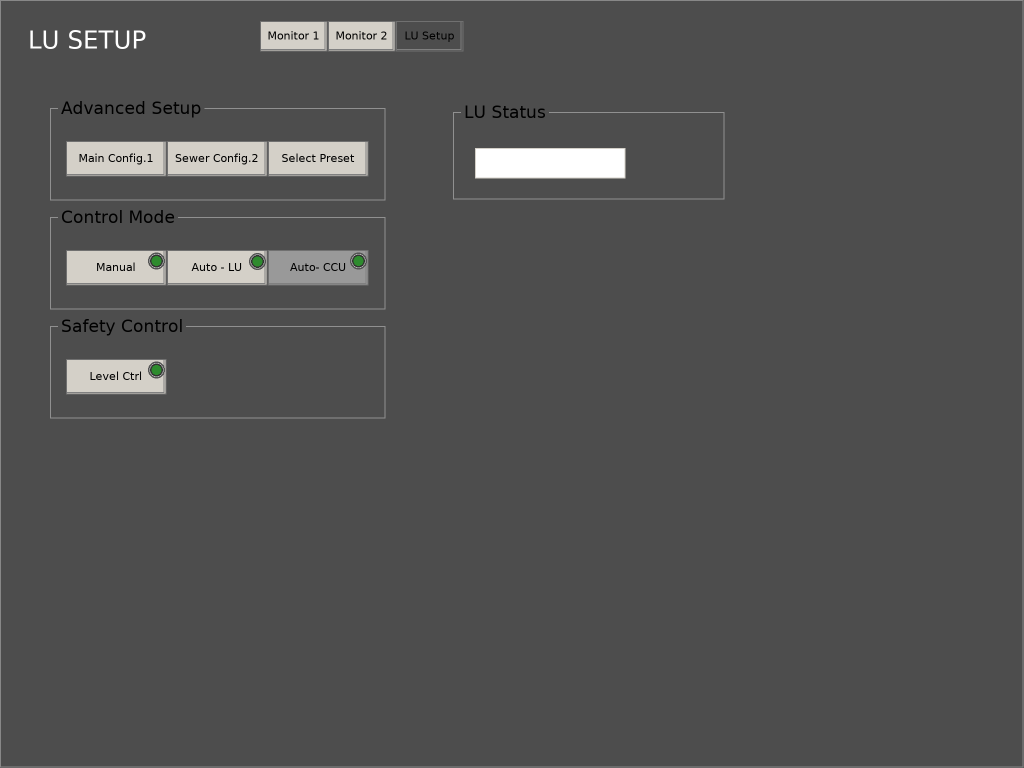
VISUALIZATION Visualization_20  // 1024x768, background image ImagePool.Background
    Label (25,25 157x30), "LU SETUP"
    GroupBox (50,209 335x100), "Control Mode"
        Button (218,41 100x35), "Auto- CCU"
            OnMouseUp: execute { GVL.MyLU.nStatus_CtrlMode := 3; }
        Button (117,41 100x35), "Auto - LU"
            OnMouseUp: execute { GVL.MyLU.nStatus_CtrlMode := 2; }
        Button (16,41 100x35), "Manual"
            OnMouseUp: execute { GVL.MyLU.nStatus_CtrlMode := 1; }
        Lamp1 (97,42 19x20), variable: GVL.MyLU.HMI_Data.ManMode, style: Lamp-Lamp1-Green
        Lamp1 (198,43 19x19), variable: GVL.MyLU.HMI_Data.LUmode, style: Lamp-Lamp1-Green
        Lamp1 (299,42 19x20), variable: GVL.MyLU.HMI_Data.CCUmode, style: Lamp-Lamp1-Green
    GroupBox (50,100 335x100), "Advanced Setup"
        Button (16,41 100x35), "Main Config.1"
            OnMouseUp:  Assign=Visualization_30, Type=Assignment
        Button (218,41 100x35), "Select Preset"
            OnMouseUp:  Assign=Visualization_40, Type=Assignment
        Button (117,41 100x35), "Sewer Config.2"
            OnMouseUp:  Assign=Visualization_31, Type=Assignment
    Button (260,21 67x30), "Monitor 1"
        OnMouseUp:  Assign=Visualization_10, Type=Assignment
    Button (328,21 67x30), "Monitor 2"
        OnMouseUp:  Assign=Visualization_11, Type=Assignment
    Button (396,21 67x30), "LU Setup"
        OnMouseUp:  Assign=Visualization_20, Type=Assignment
    GroupBox (453,104 271x95), "LU Status"
        Textfield (22,44 150x30)
    GroupBox (50,318 335x100), "Safety Control"
        Button (16,41 100x35), "Level Ctrl"
            OnMouseUp:  ToggleVariable=GVL.myLU.nStatus_LevelControl_ON
        Lamp1 (97,42 19x20), variable: GVL.MyLU.nStatus_LevelControl_ON, style: Lamp-Lamp1-Green
END_VISUALIZATION

// LocalDevice/Application/Visu_Pages/Visualization_11
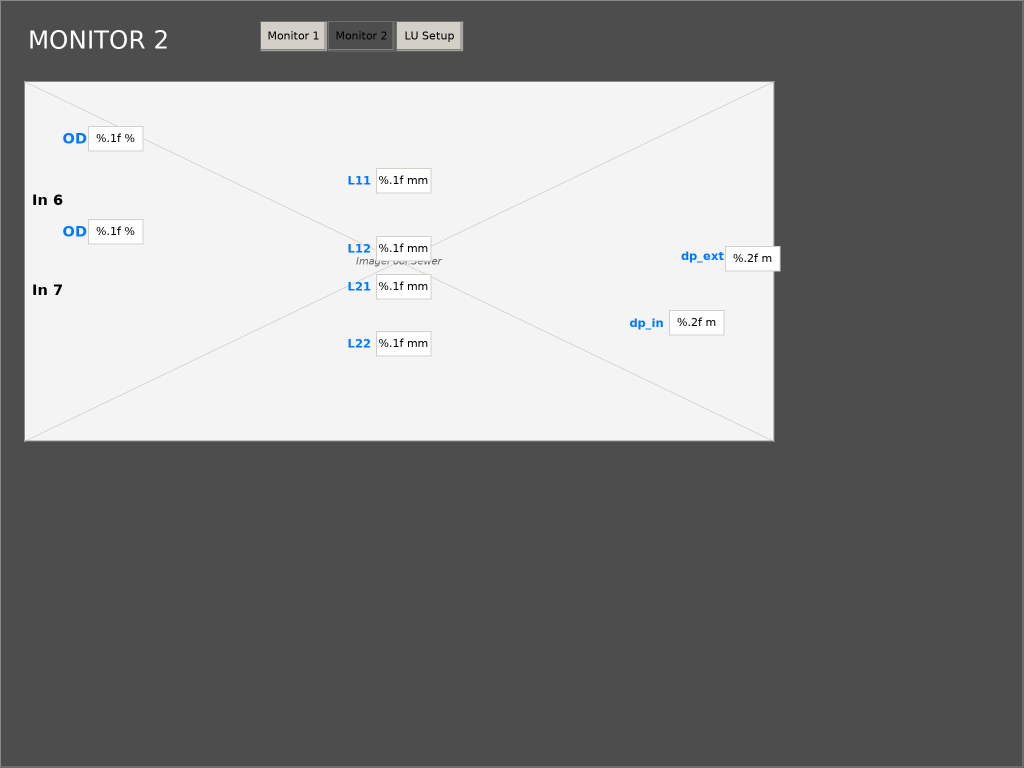
VISUALIZATION Visualization_11  // 1024x768, background image ImagePool.Background
    Label (25,25 180x30), "MONITOR 2"
    Button (260,21 67x30), "Monitor 1"
        OnMouseUp:  Assign=Visualization_10, Type=Assignment
    Button (328,21 67x30), "Monitor 2"
        OnMouseUp:  Assign=Visualization_11, Type=Assignment
    Button (396,21 67x30), "LU Setup"
        OnMouseUp:  Assign=Visualization_20, Type=Assignment
    Image (24,81 750x360), image: ImagePool.Sewer
    Label (339,168 41x25), "L11"
    Textfield (376,168 55x25), "%.1f mm", text variable: GVL.myLU.HMI_Data.L_11
    Label (339,331 41x25), "L22"
    Textfield (376,331 55x25), "%.1f mm", text variable: GVL.myLU.HMI_Data.L_22
    Label (56,126 38x25), "OD"
    Textfield (88,126 55x25), "%.1f %", text variable: GVL.myLU.HMI_Data.ValveOD_61
    Label (56,219 38x25), "OD"
    Textfield (88,219 55x25), "%.1f %", text variable: GVL.myLU.HMI_Data.ValveOD_71
    Label (339,274 41x25), "L21"
    Textfield (376,274 55x25), "%.1f mm", text variable: GVL.myLU.HMI_Data.L_21
    Label (339,236 41x25), "L12"
    Textfield (376,236 55x25), "%.1f mm", text variable: GVL.myLU.HMI_Data.L_12
    Label (626,308 41x30), "dp_in"
    Textfield (725,246 55x25), "%.2f m", text variable: GVL.myLU.HMI_Data.dP2_ex
    Label (682,241 41x30), "dp_ext"
    Textfield (669,310 55x25), "%.2f m", text variable: GVL.myLU.HMI_Data.dP2_in
    Label (18,189 59x22), "In 6"
    Label (18,279 59x22), "In 7"
END_VISUALIZATION

// LocalDevice/Application/Visu_Pages/Visualization_40
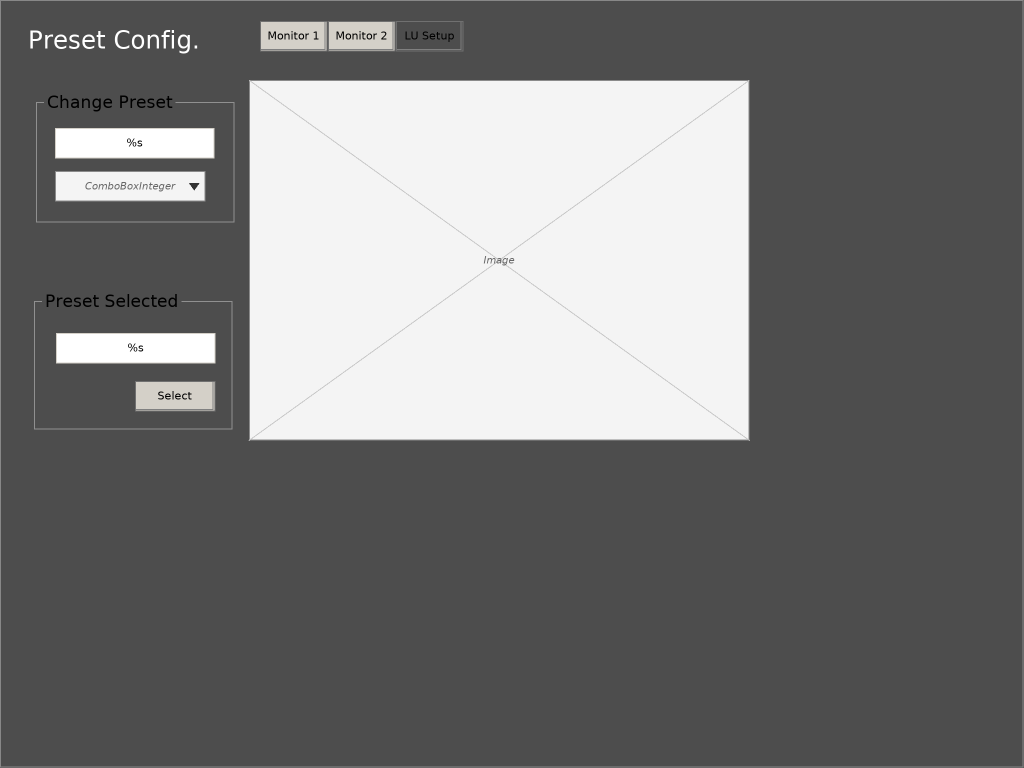
VISUALIZATION Visualization_40  // 1024x768, background image ImagePool.Background
    Label (25,25 318x30), "Preset Config."
    Button (260,21 67x30), "Monitor 1"
        OnMouseUp:  Assign=Visualization_10, Type=Assignment
    Button (328,21 67x30), "Monitor 2"
        OnMouseUp:  Assign=Visualization_11, Type=Assignment
    Button (396,21 67x30), "LU Setup"
        OnMouseUp:  Assign=Visualization_20, Type=Assignment
    Image (249,80 500x360)
        p84334746: GVL.DynamicImgID
    GroupBox (36,94 198x128), "Change Preset"
        ComboBoxInteger (19,77 150x30), variable: GVL.myLU.Idx_PresetHMI
            p1601986498: 'ImagePool_Presets'
        Textfield (19,34 159x30), "%s", text variable: GVL.myLU.PresetLU[GVL.myLU.Idx_PresetHMI].Name
    GroupBox (34,293 198x136), "Preset Selected"
        Textfield (22,40 159x30), "%s", text variable: GVL.myLU.PresetLU[GVL.myLU.Idx_Preset].Name
        Button (101,88 80x30), "Select"
            OnMouseUp: execute { GVL.myLU.Idx_Preset := GVL.myLU.Idx_PresetHMI; }
END_VISUALIZATION

// LocalDevice/Application/Visu_Pages/Visualization_31
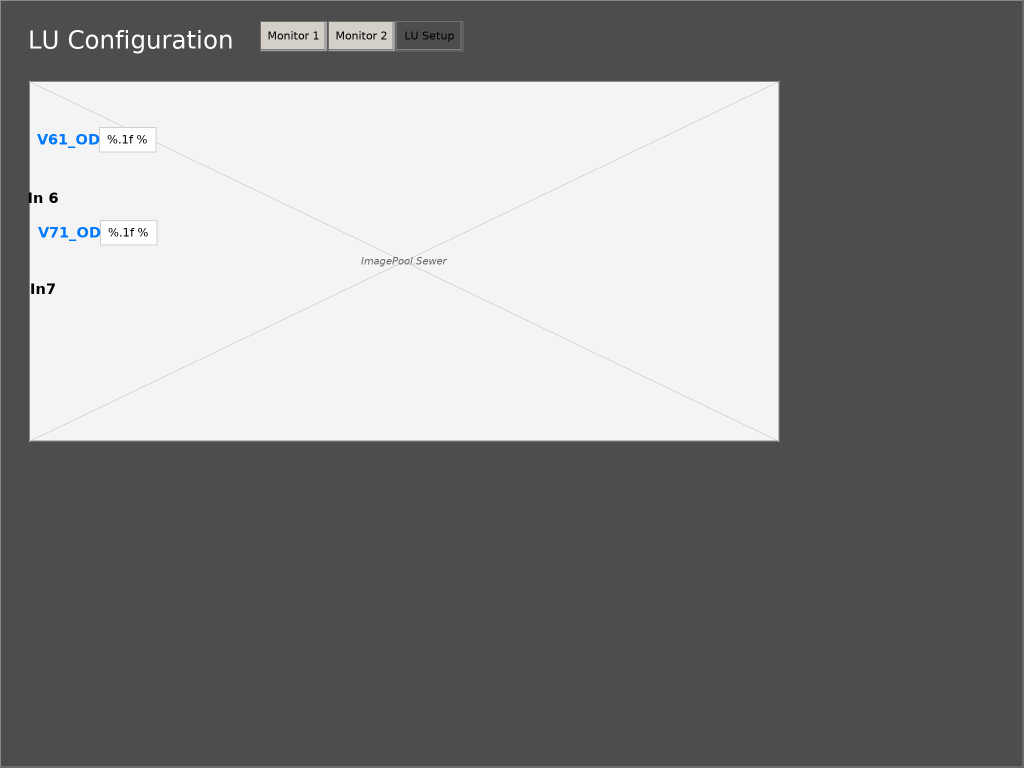
VISUALIZATION Visualization_31  // 1024x768, background image ImagePool.Background
    Image (29,81 750x360), image: ImagePool.Sewer
    Label (25,25 318x30), "LU Configuration"
    Button (260,21 67x30), "Monitor 1"
        OnMouseUp:  Assign=Visualization_10, Type=Assignment
    Button (328,21 67x30), "Monitor 2"
        OnMouseUp:  Assign=Visualization_11, Type=Assignment
    Button (396,21 67x30), "LU Setup"
        OnMouseUp:  Assign=Visualization_20, Type=Assignment
    Label (10,187 66x22), "In 6"
    Label (10,278 66x22), "In7"
    Textfield (99,127 57x25), "%.1f %", text variable: GVL.myLU.HMI_Data.ValveOD_61
        OnMouseUp: write GVL.myLU.HMI_Data.ValveOD_61_input via VisuDialogs.Numpad, min 0, max 100, format 0
    Label (41,127 55x25), "V61_OD"
    Textfield (100,220 57x25), "%.1f %", text variable: GVL.myLU.HMI_Data.ValveOD_71
        OnMouseUp: write GVL.myLU.HMI_Data.ValveOD_71_input via VisuDialogs.Numpad, min 0, max 100, format 0
    Label (42,220 55x25), "V71_OD"
END_VISUALIZATION
